// TwinCAT 3 PLC project tc_project_app
// ProgramVersion: 3.1.4023.0
// libraries:
//   Tc2_EtherCAT, * (Beckhoff Automation GmbH)
//   Tc2_MC2, * (Beckhoff Automation GmbH)
//   Tc2_MC2_Drive, * (Beckhoff Automation GmbH)
//   Tc2_Standard, * (Beckhoff Automation GmbH)
//   Tc2_SUPS, * (Beckhoff Automation GmbH)
//   Tc2_System, * (Beckhoff Automation GmbH)
//   Tc2_Utilities, * (Beckhoff Automation GmbH)
//   Tc3_MC2_AdvancedHoming, * (Beckhoff Automation GmbH)
//   Tc3_Module, * (Beckhoff Automation GmbH)
//   VisuDialogs, * (System)
// project tree:
//   DUTs/ E_RotationBrakeCheckerState.TcDUT, ST_AxisSpg.TcDUT, ST_DefaultVals.TcDUT
//   / GlobalTextList.TcGTLO (not stored), PlcTask.TcTTO, Visualization Manager.TcVMO (not stored)
//   GVLs/ GVL_APP.TcGVL, GVL_INTER.TcGVL, GVL_Safety.TcGVL
//   POUs/Application_Specific/Applications/ Application_Template.TcPOU (not stored), eState_INTER.TcDUT, eState_Vertical.TcDUT, Inclinometer.TcPOU, INTER_LOGIC.TcPOU, PLC_SAFETY_LOGIC.TcPOU, SBT_CODE_notused.TcPOU, Slit_3.TcPOU, VirtualSpeedOverrides.TcPOU
//   POUs/Application_Specific/Axes/ AXIS_NAMES.TcGVL, Axis_Template.TcPOU (not stored), Slit_West.TcPOU, Slit_North.TcPOU, Combined_Vertical.TcPOU, Horizontal_Translation.TcPOU, Slit_South.TcPOU, Slit_East.TcPOU, Vertical_Translation_Y2.TcPOU, Vertical_Translation_Y1.TcPOU, Rotation.TcPOU, Pneumatics_Template.TcPOU (not stored)
//   POUs/Application_Specific/Axes/Real axis follows/ Combined_Vertical_Virtual.TcPOU, Horizontal_Virtual.TcPOU, Rotation_Virtual.TcPOU
//   POUs/Application_Specific/Axes/Sample and Calibration/ Measurement_Angle_Offset.TcPOU, Rotation_Calibration.TcPOU, Horizontal_Calibration.TcPOU, Combined_Vertical_Calibration.TcPOU, Rotation_Sample.TcPOU, Horizontal_Sample.TcPOU, Combined_Vertical_Sample.TcPOU
//   POUs/Application_Specific/Axes/Virtuals/ Delta.TcPOU, Doff_Angled.TcPOU, Doff_Parallel.TcPOU, Drad.TcPOU, Drad_External.TcPOU, Drad_Internal.TcPOU, Dtank_Internal_Offset_Angle.TcPOU, Dtank_Length.TcPOU, Dtank_Pivot_To_Window.TcPOU, Measurement_Angle.TcPOU, Tau.TcPOU
//   POUs/ MAIN.TcPOU
//   tc_mca_std_lib/DUTs/Axis_Structures/ ST_AxisConfig.TcDUT (not stored), ST_AxisControl.TcDUT (not stored), ST_AxisDescription.TcDUT, ST_AxisError.TcDUT (not stored), ST_AxisInputs.TcDUT (not stored), ST_AxisPersistent.TcDUT (not stored), ST_AxisSafety.TcDUT (not stored), ST_AxisStatus.TcDUT, ST_AxisStruct.TcDUT, ST_GearAxis.TcDUT (not stored)
//   tc_mca_std_lib/DUTs/ E_AxisParameters.TcTLEO (not stored), E_HomingRoutines.TcTLEO, E_AxisParameters.TcTLEO (not stored), E_MonitoringLedFunction.TcDUT (not stored), E_MotorTypeClass.TcDUT, E_EncoderTypeClass.TcDUT, E_HomeSwitchTypeClass.TcDUT, E_RestorePosition.TcDUT (not stored), I_Axis.TcIO (not stored), E_SlitPairStatesV2.TcDUT (not stored), E_SlitPairStates.TcDUT (not stored), ST_MonitoringAlarm.TcDUT (not stored), E_MotionFunctions.TcDUT (not stored), ST_McStatus.TcDUT (not stored)
//   tc_mca_std_lib/DUTs/Pneumatics/ E_PneumaticAxisErrors.TcDUT (not stored), E_PneumaticMode.TcDUT (not stored), ST_PneumaticAxisControl.TcDUT (not stored), ST_PneumaticAxisConfig.TcDUT (not stored), ST_PneumaticAxisInputs.TcDUT (not stored), ST_PneumaticAxisOutputs.TcDUT (not stored), ST_PneumaticAxisStatus.TcDUT (not stored), ST_PneumaticAxisStruct.TcDUT (not stored)
//   tc_mca_std_lib/DUTs/Safety Status/ E_SafetyFbState.TcDUT, E_SafetyFbType.TcDUT, E_SafetyGroupState.TcDUT, E_SafetyDevices.TcDUT (not stored), FB_SafeFBDiag.TcPOU, ST_SafetyAliasInput.TcDUT, ST_SafetyData.TcDUT, ST_SafetyDevice.TcDUT (not stored), ST_SafetyFB.TcDUT, ST_SafetyGroup.TcDUT, ST_SafetyAliasOutput.TcDUT, ST_SafetyProject.TcDUT
//   tc_mca_std_lib/GVLs/ GVL.TcGVL
//   tc_mca_std_lib/POUs/ FB_ESSMonitoring.TcPOU
//   tc_mca_std_lib/POUs/Motion/ FB_Axis.TcPOU, FB_SlitPair.TcPOU (not stored), FB_SlitPairV2.TcPOU (not stored)
//   tc_mca_std_lib/POUs/Motion/Homing/ FB_Homing.TcPOU (not stored)
//   tc_mca_std_lib/POUs/Pneumatics/ FB_PneumaticAxis.TcPOU (not stored)
//   tc_mca_std_lib/VISUs/ languageSupport.TcTLO (not stored), MainVisu.TcVIS, ParameterTextList.TcTLO (not stored), PneumaticsVisu.TcVIS (not stored)
// real-time tasks:
//   TASK PlcTask: cycle T#2ms, priority 10, ADS port 351
// motion (NC):
//   TASK NC-Task 1 SAF: cycle T#2ms, priority 4, ADS port 501
//   TASK NC-Task 1 SVB: cycle T#10ms, priority 8, ADS port 511
//   AXIS M1 - South (id 1)
//     Dynamic: AccelerationMaximum=50, DecelerationMaximum=50, Acceleration=25, Deceleration=25, Jerk=60
//     Velo: RefSearch=0.5, RefSync=0.5, SlowManual=0.5, FastManual=1, Maximum=1.2
//     OtherSettings: AllowMotionCmdToSlave=true, DataPersistence=true
//     encoder EncType=4
//       EncPara: ScaleFactorNumerator=0.001, MaxCount=#x0000ffff
//         Inc: RefMode=2, RefSoftSyncMask=#x0000ffff
//     drive DrvType=24
//       DrvPara: Inverse=true
//         Analog: VeloReferenz=2, TorqueSetpointScale=10, ScaleFactorActTorque=0.1
//         TimeComp: TaskDelayCycles=1
//     controller CtrType=1
//       CtrPara: PriorControlFactor=1
//         Observer: BandWidth=20
//   AXIS M2 - North (id 2)
//     Dynamic: AccelerationMaximum=50, DecelerationMaximum=50, Acceleration=25, Deceleration=25, Jerk=60
//     Velo: RefSearch=0.5, RefSync=0.5, SlowManual=0.5, FastManual=1, Maximum=1.2
//     OtherSettings: AllowMotionCmdToSlave=true, DataPersistence=true
//     encoder EncType=4
//       EncPara: ScaleFactorNumerator=0.001, MaxCount=#x0000ffff
//         Inc: RefMode=2, RefSoftSyncMask=#x0000ffff
//     drive DrvType=24
//       Analog: VeloReferenz=2, TorqueSetpointScale=10, ScaleFactorActTorque=0.1
//       TimeComp: TaskDelayCycles=1
//     controller CtrType=1
//       CtrPara: PriorControlFactor=1
//         Observer: BandWidth=20
//   AXIS M3 - West (id 3)
//     Dynamic: AccelerationMaximum=50, DecelerationMaximum=50, Acceleration=25, Deceleration=25, Jerk=60
//     Velo: RefSearch=0.5, RefSync=0.5, SlowManual=0.5, FastManual=1, Maximum=1.2
//     OtherSettings: AllowMotionCmdToSlave=true, DataPersistence=true
//     encoder EncType=4
//       EncPara: ScaleFactorNumerator=0.001, MaxCount=#x0000ffff
//         Inc: RefMode=2, RefSoftSyncMask=#x0000ffff
//     drive DrvType=24
//       DrvPara: Inverse=true
//         Analog: VeloReferenz=2, TorqueSetpointScale=10, ScaleFactorActTorque=0.1
//         TimeComp: TaskDelayCycles=1
//     controller CtrType=1
//       CtrPara: PriorControlFactor=1
//         Observer: BandWidth=20
//   AXIS M4 - East (id 4)
//     Dynamic: AccelerationMaximum=50, DecelerationMaximum=50, Acceleration=25, Deceleration=25, Jerk=60
//     Velo: RefSearch=0.5, RefSync=0.5, SlowManual=0.5, FastManual=1, Maximum=1.2
//     OtherSettings: AllowMotionCmdToSlave=true, DataPersistence=true
//     encoder EncType=4
//       EncPara: ScaleFactorNumerator=0.001, MaxCount=#x0000ffff
//         Inc: RefMode=2, RefSoftSyncMask=#x0000ffff
//     drive DrvType=24
//       Analog: VeloReferenz=2, TorqueSetpointScale=10, ScaleFactorActTorque=0.1
//       TimeComp: TaskDelayCycles=1
//     controller CtrType=1
//       CtrPara: PriorControlFactor=1
//         Observer: BandWidth=20
//   AXIS Rotation (id 5)
//     General: UnitName=°
//     Dynamic: AccelerationMaximum=19997.325, DecelerationMaximum=19997.325, Acceleration=30, Deceleration=30, Jerk=35.7075
//     Velo: RefSearch=0.07935, RefSync=0.07935, SlowManual=0.05, FastManual=0.6, Fast=7.935, Maximum=8
//     OtherSettings: AllowMotionCmdToSlave=true, DataPersistence=true
//     encoder EncType=19
//       EncPara: ScaleFactorNumerator=360, ScaleFactorDenominator=1761607680, Offset=-201.549349812099, MaxCount=#xffffffff, ReferenceSystem=1
//     drive DrvType=16
//       DrvPara: MaxCount=#xffffffff, DriveControlDWord=#x00020100
//         Analog: VeloReferenz=8.7285, VeloScale=71.5255737304688, TorqueSetpointScale=10, ScaleFactorActTorque=0.1
//         TimeComp: TaskDelayCycles=1
//     controller CtrType=1
//       CtrPara: PriorControlFactor=1
//         PosDiffControl: Range=4
//         Observer: BandWidth=20
//   AXIS Horizontal Z Translation (id 6)
//     Dynamic: Acceleration=34.773, Deceleration=34.773, Jerk=104.319
//     Velo: RefSearch=0.23182, RefSync=0.23182, SlowManual=2, FastManual=4, Fast=23.182, Maximum=20
//     PositionAreaControl: Enable=false
//     TargetPosControl: Range=0.005, Time=0.04
//     OtherSettings: AllowMotionCmdToSlave=true
//     encoder EncType=19
//       EncPara: ScaleFactorNumerator=0.001, ScaleFactorDenominator=1000, Offset=2359.51, Inverse=true, MaxCount=#xffffffff, ReferenceSystem=1
//         Inc: RefSoftSyncMask=#x0007a11f
//     drive DrvType=16
//       DrvPara: Inverse=true, MaxCount=#xffffffff, DriveControlDWord=#x00020000
//         Analog: VeloReferenz=25.5002, VeloScale=71.5255737304688, TorqueSetpointScale=10, ScaleFactorActTorque=0.1
//         TimeComp: TaskDelayCycles=1
//     controller CtrType=1
//       CtrPara: PriorControlFactor=1
//         PosDiffControl: Enable=false
//         Observer: BandWidth=20
//   AXIS Vertical Y1 (id 7) // ACTUALLY Y?
//     Dynamic: Acceleration=10, Deceleration=10, Jerk=40
//     Velo: RefSearch=0.37029, RefSync=0.37029, SlowManual=5, FastManual=30, Fast=37.029, Maximum=32
//     PositionAreaControl: Enable=false
//     TargetPosControl: Range=0.01
//     OtherSettings: AllowMotionCmdToSlave=true
//     encoder EncType=19
//       EncPara: ScaleFactorNumerator=0.001, ScaleFactorDenominator=1000, Offset=91.510823, Inverse=true, MaxCount=#xffffffff, ReferenceSystem=1, EncPositionSource=1
//         Inc: RefSoftSyncMask=#x000f423f
//     drive DrvType=16
//       DrvPara: Inverse=true, MaxCount=#xffffffff, DriveControlDWord=#x00020000
//         Analog: VeloReferenz=40.7319, VeloScale=71.5255737304688, TorqueSetpointScale=10, ScaleFactorActTorque=0.1
//         TimeComp: TaskDelayCycles=1
//     controller CtrType=1
//       CtrPara: PriorControlFactor=1
//         PID: PosKp=2
//         Observer: BandWidth=20
//   AXIS Vertical Y2 (id 8)
//     Dynamic: Acceleration=10, Deceleration=10, Jerk=40
//     Velo: RefSearch=0.37029, RefSync=0.37029, SlowManual=5, FastManual=30, Fast=37.029, Maximum=32
//     PositionAreaControl: Enable=false
//     TargetPosControl: Range=0.01
//     OtherSettings: AllowMotionCmdToSlave=true
//     encoder EncType=19
//       EncPara: ScaleFactorNumerator=0.001, ScaleFactorDenominator=1000, Offset=93.490647, MaxCount=#xffffffff, ReferenceSystem=1
//         Inc: RefSoftSyncMask=#x000f423f
//     drive DrvType=16
//       DrvPara: MaxCount=#xffffffff, DriveControlDWord=#x00020000
//         Analog: VeloReferenz=40.7319, VeloScale=71.5255737304688, TorqueSetpointScale=10, ScaleFactorActTorque=0.1
//         TimeComp: TaskDelayCycles=1
//     controller CtrType=1
//       CtrPara: PriorControlFactor=1
//         PID: PosKp=2
//         Observer: BandWidth=20
//   AXIS RotExtra (id 31)
//     OtherSettings: AllowMotionCmdToSlave=true
//     encoder EncType=16
//       EncPara: ScaleFactorNumerator=360, ScaleFactorDenominator=1761607680, MaxCount=#xffffffff
//     drive DrvType=5
//       Analog: TorqueSetpointScale=10, ScaleFactorActTorque=0.1
//       TimeComp: TaskDelayCycles=1
//     controller CtrType=1
//       CtrPara: PriorControlFactor=1
//         Observer: BandWidth=20
//   AXIS Detector Tank Internal Offset Angle (id 14)
//     OtherSettings: AllowMotionCmdToSlave=true
//     encoder EncType=16
//       EncPara: ScaleFactorNumerator=1e-05, MaxCount=#xffffffff, ReferenceSystem=1
//     drive DrvType=5
//       Analog: TorqueSetpointScale=10, ScaleFactorActTorque=0.1
//       TimeComp: TaskDelayCycles=1
//     controller CtrType=1
//       CtrPara: PriorControlFactor=1
//         Observer: BandWidth=20
//   AXIS Delta (id 17)
//     OtherSettings: AllowMotionCmdToSlave=true
//     encoder EncType=16
//       EncPara: ScaleFactorNumerator=1e-05, MaxCount=#xffffffff, ReferenceSystem=1
//     drive DrvType=5
//       Analog: TorqueSetpointScale=10, ScaleFactorActTorque=0.1
//       TimeComp: TaskDelayCycles=1
//     controller CtrType=1
//       CtrPara: PriorControlFactor=1
//         Observer: BandWidth=20
//   AXIS Tau (id 18)
//     OtherSettings: AllowMotionCmdToSlave=true
//     encoder EncType=16
//       EncPara: ScaleFactorNumerator=1e-05, MaxCount=#xffffffff, ReferenceSystem=1
//     drive DrvType=5
//       Analog: TorqueSetpointScale=10, ScaleFactorActTorque=0.1
//       TimeComp: TaskDelayCycles=1
//     controller CtrType=1
//       CtrPara: PriorControlFactor=1
//         Observer: BandWidth=20
//   AXIS Detector Radius External (id 10)
//     OtherSettings: AllowMotionCmdToSlave=true
//     encoder EncType=16
//       EncPara: ScaleFactorNumerator=1e-05, MaxCount=#xffffffff, ReferenceSystem=1
//     drive DrvType=5
//       Analog: TorqueSetpointScale=10, ScaleFactorActTorque=0.1
//     controller CtrType=1
//       CtrPara: PriorControlFactor=1
//         Observer: BandWidth=20
//   AXIS Detector Radius Internal (id 11)
//     OtherSettings: AllowMotionCmdToSlave=true
//     encoder EncType=16
//       EncPara: ScaleFactorNumerator=1e-05, MaxCount=#xffffffff, ReferenceSystem=1
//     drive DrvType=5
//       Analog: TorqueSetpointScale=10, ScaleFactorActTorque=0.1
//     controller CtrType=1
//       CtrPara: PriorControlFactor=1
//         Observer: BandWidth=20
//   AXIS Combined Vertical (id 9)
//     Dynamic: Acceleration=60, Deceleration=60, Jerk=40
//     Velo: RefSearch=0.37029, RefSync=0.37029, SlowManual=10, FastManual=15, Fast=37.029, Maximum=30
//     PositionAreaControl: Enable=false
//     TargetPosControl: Range=0.005, Time=0.2
//     OtherSettings: AllowMotionCmdToSlave=true
//     encoder EncType=1
//       EncPara: ScaleFactorNumerator=0.001, ScaleFactorDenominator=1000, Offset=67.6442, Inverse=true, ReferenceSystem=1
//     drive DrvType=5
//       DrvPara: Inverse=true
//         Analog: VeloReferenz=40.7319, TorqueSetpointScale=10, ScaleFactorActTorque=0.1
//         TimeComp: TaskDelayCycles=1
//     controller CtrType=1
//       CtrPara: PriorControlFactor=0.8
//         Observer: BandWidth=20
//   AXIS Horizontal Virtual (id 30)
//     OtherSettings: AllowMotionCmdToSlave=true
//     encoder EncType=16
//       EncPara: ScaleFactorNumerator=1e-05, MaxCount=#xffffffff, ReferenceSystem=1
//     drive DrvType=5
//       Analog: TorqueSetpointScale=10, ScaleFactorActTorque=0.1
//       TimeComp: TaskDelayCycles=1
//     controller CtrType=1
//       CtrPara: PriorControlFactor=1
//         Observer: BandWidth=20
//   AXIS Rotation Virtual (id 23)
//     OtherSettings: AllowMotionCmdToSlave=true
//     encoder EncType=16
//       EncPara: ScaleFactorNumerator=1e-05, MaxCount=#xffffffff, ReferenceSystem=1
//     drive DrvType=5
//       Analog: TorqueSetpointScale=10, ScaleFactorActTorque=0.1
//       TimeComp: TaskDelayCycles=1
//     controller CtrType=1
//       CtrPara: PriorControlFactor=1
//         Observer: BandWidth=20
//   AXIS Combined Vertical Virtual (id 27)
//     OtherSettings: AllowMotionCmdToSlave=true
//     encoder EncType=16
//       EncPara: ScaleFactorNumerator=1e-05, MaxCount=#xffffffff, ReferenceSystem=1
//     drive DrvType=5
//       Analog: TorqueSetpointScale=10, ScaleFactorActTorque=0.1
//       TimeComp: TaskDelayCycles=1
//     controller CtrType=1
//       CtrPara: PriorControlFactor=1
//         Observer: BandWidth=20
//   AXIS Detector Tank Length (id 15)
//     Dynamic: Acceleration=20, Deceleration=20, Jerk=50
//     Velo: SlowManual=5, FastManual=10
//     OtherSettings: AllowMotionCmdToSlave=true
//     encoder EncType=1
//     drive DrvType=5
//       Analog: TorqueSetpointScale=10, ScaleFactorActTorque=0.1
//       TimeComp: TaskDelayCycles=1
//     controller CtrType=1
//       CtrPara: PriorControlFactor=1
//         Observer: BandWidth=20
//   AXIS Detector Tank Pivot To Window (id 16)
//     Dynamic: Acceleration=20, Deceleration=20, Jerk=50
//     Velo: SlowManual=5, FastManual=10
//     OtherSettings: AllowMotionCmdToSlave=true
//     encoder EncType=1
//     drive DrvType=5
//       Analog: TorqueSetpointScale=10, ScaleFactorActTorque=0.1
//       TimeComp: TaskDelayCycles=1
//     controller CtrType=1
//       CtrPara: PriorControlFactor=1
//         Observer: BandWidth=20
//   AXIS Rotation Calibration (id 22)
//     General: UnitName=°
//     Dynamic: Acceleration=0.5, Deceleration=0.5, Jerk=30
//     Velo: RefSearch=0.55548, RefSync=0.55548, SlowManual=0.25, FastManual=0.375, Fast=55.543, Maximum=55.543
//     TargetPosControl: Range=0.005
//     OtherSettings: AllowMotionCmdToSlave=true, DataPersistence=true
//     encoder EncType=1
//       EncPara: ScaleFactorNumerator=360, ScaleFactorDenominator=251658240, Offset=10.2575826644897, ToleranceWndModuloStart=10
//     drive DrvType=5
//       Analog: VeloReferenz=61.0973, TorqueSetpointScale=10, ScaleFactorActTorque=0.1
//       TimeComp: TaskDelayCycles=1
//     controller CtrType=1
//       CtrPara: PriorControlFactor=1
//         PID: PosKp=2
//         Observer: BandWidth=20
//   AXIS Combined Vertical Calibration (id 25)
//     Dynamic: Acceleration=20, Deceleration=20, Jerk=50
//     Velo: SlowManual=5, FastManual=10, Fast=37.029, Maximum=37.029
//     PositionAreaControl: Enable=false
//     TargetPosControl: Range=0.005, Time=0.2
//     OtherSettings: AllowMotionCmdToSlave=true
//     encoder EncType=1
//       EncPara: ScaleFactorNumerator=0.001, ScaleFactorDenominator=1000, Offset=182.9435, Inverse=true, ReferenceSystem=1
//     drive DrvType=5
//       DrvPara: Inverse=true
//         Analog: VeloReferenz=40.7319, TorqueSetpointScale=10, ScaleFactorActTorque=0.1
//         TimeComp: TaskDelayCycles=1
//     controller CtrType=1
//       CtrPara: PriorControlFactor=0.8
//         Observer: BandWidth=20
//   AXIS Horizontal Calibration (id 28)
//     Dynamic: Acceleration=20, Deceleration=20, Jerk=50
//     Velo: SlowManual=5, FastManual=10, Fast=23.182, Maximum=23.182
//     PositionAreaControl: Enable=false
//     TargetPosControl: Range=0.005, Time=0.04
//     OtherSettings: AllowMotionCmdToSlave=true
//     encoder EncType=1
//       EncPara: ScaleFactorNumerator=5, ScaleFactorDenominator=10485760, Offset=2359.51, ModuloFactor=100000000, Inverse=true, EncPositionSource=1
//     drive DrvType=5
//       DrvPara: Inverse=true
//         Analog: VeloReferenz=25.5002, TorqueSetpointScale=10, ScaleFactorActTorque=0.1
//         TimeComp: TaskDelayCycles=1
//     controller CtrType=1
//       CtrPara: PriorControlFactor=1
//         PID: PosKp=2
//         Observer: BandWidth=20
//   AXIS Detector Offset Angled (id 12)
//     Dynamic: Acceleration=0.5, Deceleration=0.5, Jerk=30
//     Velo: RefSearch=0.55548, RefSync=0.55548, SlowManual=0.25, FastManual=0.375
//     OtherSettings: AllowMotionCmdToSlave=true
//     encoder EncType=1
//     drive DrvType=5
//       Analog: TorqueSetpointScale=10, ScaleFactorActTorque=0.1
//       TimeComp: TaskDelayCycles=1
//     controller CtrType=1
//       CtrPara: PriorControlFactor=1
//         Observer: BandWidth=20
//   AXIS Detector Offset Parallel (id 13)
//     Dynamic: Acceleration=0.5, Deceleration=0.5, Jerk=30
//     Velo: RefSearch=0.55548, RefSync=0.55548, SlowManual=5, FastManual=10
//     OtherSettings: AllowMotionCmdToSlave=true
//     encoder EncType=1
//     drive DrvType=5
//       Analog: TorqueSetpointScale=10, ScaleFactorActTorque=0.1
//       TimeComp: TaskDelayCycles=1
//     controller CtrType=1
//       CtrPara: PriorControlFactor=1
//         Observer: BandWidth=20
//   AXIS Detector Radius (id 19)
//     Dynamic: Acceleration=20, Deceleration=20, Jerk=50
//     Velo: SlowManual=5, FastManual=10
//     OtherSettings: AllowMotionCmdToSlave=true
//     encoder EncType=1
//       EncPara: ScaleFactorNumerator=1e-06
//     drive DrvType=5
//       Analog: TorqueSetpointScale=10, ScaleFactorActTorque=0.1
//       TimeComp: TaskDelayCycles=1
//     controller CtrType=1
//       CtrPara: PriorControlFactor=1
//         Observer: BandWidth=20
//   AXIS Measurement Angle (id 20)
//     Dynamic: AccelerationMaximum=600, DecelerationMaximum=600, Acceleration=0.3, Deceleration=0.3, Jerk=10
//     Velo: RefSearch=0.55548, RefSync=0.55548, SlowManual=0.25, FastManual=0.375, Maximum=2
//     OtherSettings: AllowMotionCmdToSlave=true
//     encoder EncType=1
//       EncPara: ScaleFactorNumerator=1e-06
//     drive DrvType=5
//       Analog: TorqueSetpointScale=10, ScaleFactorActTorque=0.1
//       TimeComp: TaskDelayCycles=1
//     controller CtrType=1
//       CtrPara: PriorControlFactor=1
//         Observer: BandWidth=20
//   AXIS Measurement Angle Offset (id 21)
//     Dynamic: AccelerationMaximum=600, DecelerationMaximum=600, Acceleration=0.5, Deceleration=0.5, Jerk=30
//     Velo: RefSearch=0.55548, RefSync=0.55548, SlowManual=0.25, FastManual=0.375, Maximum=0.6
//     OtherSettings: AllowMotionCmdToSlave=true
//     encoder EncType=1
//       EncPara: ScaleFactorNumerator=1e-06
//     drive DrvType=5
//       Analog: TorqueSetpointScale=10, ScaleFactorActTorque=0.1
//       TimeComp: TaskDelayCycles=1
//     controller CtrType=1
//       CtrPara: PriorControlFactor=1
//         Observer: BandWidth=20
//   AXIS Rotation Sample (id 24)
//     General: UnitName=°
//     Dynamic: Acceleration=0.5, Deceleration=0.5, Jerk=30
//     Velo: RefSearch=0.55548, RefSync=0.55548, SlowManual=0.25, FastManual=0.375, Fast=55.543, Maximum=55.543
//     OtherSettings: AllowMotionCmdToSlave=true, DataPersistence=true
//     encoder EncType=1
//       EncPara: ScaleFactorNumerator=360, ScaleFactorDenominator=251658240, Offset=10.2575826644897, ToleranceWndModuloStart=10
//     drive DrvType=5
//       Analog: VeloReferenz=61.0973, TorqueSetpointScale=10, ScaleFactorActTorque=0.1
//       TimeComp: TaskDelayCycles=1
//     controller CtrType=1
//       CtrPara: PriorControlFactor=1
//         PID: PosKp=2
//         Observer: BandWidth=20
//   AXIS Combined Vertical Sample (id 26)
//     Dynamic: Acceleration=20, Deceleration=20, Jerk=50
//     Velo: SlowManual=5, FastManual=10, Fast=37.029, Maximum=37.029
//     PositionAreaControl: Enable=false
//     TargetPosControl: Range=0.005, Time=0.2
//     OtherSettings: AllowMotionCmdToSlave=true
//     encoder EncType=1
//       EncPara: ScaleFactorNumerator=0.001, ScaleFactorDenominator=1000, Inverse=true, ReferenceSystem=1
//     drive DrvType=5
//       DrvPara: Inverse=true
//         Analog: VeloReferenz=40.7319, TorqueSetpointScale=10, ScaleFactorActTorque=0.1
//         TimeComp: TaskDelayCycles=1
//     controller CtrType=1
//       CtrPara: PriorControlFactor=0.8
//         Observer: BandWidth=20
//   AXIS Horizontal Sample (id 29)
//     Dynamic: Acceleration=34.773, Deceleration=34.773, Jerk=104.319
//     Velo: RefSearch=0.23182, RefSync=0.23182, SlowManual=5, FastManual=10, Fast=23.182, Maximum=23.182
//     PositionAreaControl: Enable=false
//     TargetPosControl: Range=0.005, Time=0.04
//     OtherSettings: AllowMotionCmdToSlave=true
//     encoder EncType=1
//       EncPara: ScaleFactorNumerator=5, ScaleFactorDenominator=10485760, Offset=2359.51, ModuloFactor=100000000, Inverse=true, EncPositionSource=1
//     drive DrvType=5
//       DrvPara: Inverse=true
//         Analog: VeloReferenz=25.5002, TorqueSetpointScale=10, ScaleFactorActTorque=0.1
//         TimeComp: TaskDelayCycles=1
//     controller CtrType=1
//       CtrPara: PriorControlFactor=1
//         PID: PosKp=2
//         Observer: BandWidth=20
// I/O:
//   DEVICE Device 1 (EtherCAT), AmsNetId 5.119.206.217.2.1
//     Term 1 (EK1200) [EK1200-5000 EtherCAT Power supply (2A E-Bus)]
//       Term 2 (EL6070-0033) [EL6070-0033 1Ch. Licence key terminal, individual licences]
//       Term 3 (EL3004) [EL3004 4Ch. Ana. Input +/-10V]
//       Term 39 (EL3621-0020) [EL3621-0020 1Ch. Ana. Input 4-20 mA, Diff. 24bit, High Precision, calibrated]
//       Term 5 (EL4004) [EL4004 4Ch. Ana. Output 0-10V, 12bit]
//       Term 6 (EL4024) [EL4024 4Ch. Ana. Output 4-20mA, 12bit]
//       Term 7 (EL1008) [EL1008 8Ch. Dig. Input 24V, 3ms]
//       Term 8 (EL2008) [EL2008 8Ch. Dig. Output 24V, 0.5A]
//       Term 9 (EL1008) [EL1008 8Ch. Dig. Input 24V, 3ms]
//       EL10088-(03) [EL1008 8Ch. Dig. Input 24V, 3ms]
//       Term 11 (EL6688) [EL6688 - External Synchronisation Interface (IEEE1588)]
//       Term 12 (EL9410) [EL9410 E-Bus Power Supplier  (Diagnostics)]
//       EL2008-(02) [EL2008 8Ch. Dig. Output 24V, 0.5A]
//       EL2008-(03) [EL2008 8Ch. Dig. Output 24V, 0.5A]
//       Term 50 (EL3152) [EL3152 2Ch. Ana Input 4-20mA]
//       Term 16 (EK1110) [EK1110 EtherCAT extension]
//     Term 17 (EK1100) [EK1100 EtherCAT Coupler (2A E-Bus)]
//       Term 18 (EL5101) [EL5101 1Ch. Inc. Encoder 5V]
//       Term 19 (EL5101) [EL5101 1Ch. Inc. Encoder 5V]
//       Term 20 (EL5101) [EL5101 1Ch. Inc. Encoder 5V]
//       Term 21 (EL5101) [EL5101 1Ch. Inc. Encoder 5V]
//       Term 36 (EL9011) [EL9011 End Terminal]
//     Term 22 (EK1100) [EK1100 EtherCAT Coupler (2A E-Bus)]
//       Term 23 (EL7047) [EL7047 1Ch. Stepper motor output stage (50V, 5A)]
//       Term 24 (EL7047) [EL7047 1Ch. Stepper motor output stage (50V, 5A)]
//       Term 25 (EL7047) [EL7047 1Ch. Stepper motor output stage (50V, 5A)]
//       Term 26 (EL7047) [EL7047 1Ch. Stepper motor output stage (50V, 5A)]
//       Term 37 (EL9011) [EL9011 End Terminal]
//     Term 27 (EK1100) [EK1100 EtherCAT Coupler (2A E-Bus)]
//       EL6910-(04) [EL6910, TwinSAFE PLC]
//       EL2904-(06) [EL2904, 4 Ch. Safety Output 24V, 0.5A, TwinSAFE]
//         modules: Module 1 (FSOES), Module 2 (DO)
//       EL1904-(06) [EL1904, 4 Ch. Safety Input 24V, TwinSAFE]
//         modules: Module 1 (FSOES)
//       EL1904-(07) [EL1904, 4 Ch. Safety Input 24V, TwinSAFE]
//         modules: Module 1 (FSOES)
//       EL1904-(08) [EL1904, 4 Ch. Safety Input 24V, TwinSAFE]
//         modules: Module 1 (FSOES)
//       EL1904-(09) [EL1904, 4 Ch. Safety Input 24V, TwinSAFE]
//         modules: Module 1 (FSOES)
//       EL1904-(10) [EL1904, 4 Ch. Safety Input 24V, TwinSAFE]
//         modules: Module 1 (FSOES)
//       EL1904-(11) [EL1904, 4 Ch. Safety Input 24V, TwinSAFE]
//         modules: Module 1 (FSOES)
//       EL2912-(07) [EL2912, 2Ch. Safety Output 24V, 2A, TwinSAFE]
//         modules: Module 1 (FSOE), Module 2 (FSOUT), Module 3 (DEVICEIO), Module 4 (FSLOGIC)
//       Term 80 (EL9410) [EL9410 E-Bus Power Supplier  (Diagnostics)]
//       EL1904-(12) [EL1904, 4 Ch. Safety Input 24V, TwinSAFE]
//         modules: Module 1 (FSOES)
//       EL1904-(13) [EL1904, 4 Ch. Safety Input 24V, TwinSAFE]
//         modules: Module 1 (FSOES)
//       EL2904-(08) [EL2904, 4 Ch. Safety Output 24V, 0.5A, TwinSAFE]
//         modules: Module 1 (FSOES), Module 2 (DO)
//       EL2904-(09) [EL2904, 4 Ch. Safety Output 24V, 0.5A, TwinSAFE]
//         modules: Module 1 (FSOES), Module 2 (DO)
//       Term 38 (EL9011) [EL9011 End Terminal]
//     Term 70 (AX8640-0000-0103) [AX8640-0000-0103]
//       Drive 71 (AX8206-0210-0104) [AX8206-0210-0104 (2Ch. 6A servo axis, safe-motion, multi-FB)]
//         modules: Device, Device, Device, Device, Device, Device, Device, Device, Device, Device, Device (Safety), Device, Device, Device, Device, Device, Device, Device, Device, Device, Device, Device, Device, Device, Device, Device, Device, Device, Device, Device, Device, Ch A, Ch A, Ch A, Ch A, Ch A, Ch A, Ch A, Ch A, Ch A, Ch A, Ch A, Ch A, Ch A, Ch A, Ch A, Ch A, Ch A, Ch A, Ch A, Ch A, Ch A, Ch A, Ch A, Ch A, Ch A, Ch A, Ch A, Ch B, Ch B, Ch B, Ch B, Ch B, Ch B, Ch B, Ch B, Ch B, Ch B, Ch B, Ch B, Ch B, Ch B, Ch B, Ch B, Ch B, Ch B, Ch B, Ch B, Ch B, Ch B, Ch B, Ch B, Ch B, Ch B, Ch B
//         startup 12992:1 := 414D383035332D78477831 // Ch A Motor parameters / Configured motor type
//         startup 24768:0 := FEFF // Ch A Interpolation sub mode select
//         startup 13000:5 := 0200 // Ch A Motor thermal model / Reaction
//         startup 13000:6 := 0000C841 // Ch A Motor thermal model / Partial fraction factor
//         startup 12992:12 := 0000FA44 // Ch A Motor parameters / Motor rated speed
//         startup 12992:13 := 73681F41 // Ch A Motor parameters / Motor rated torque
//         startup 24694:0 := 9D2C0000 // Ch A Motor standstill torque
//         startup 24800:0 := D007 // Ch A Positive torque/force limit value
//         startup 24801:0 := D007 // Ch A Negative torque/force limit value
//         startup 12288:6 := 4158383230362D303231302D30303030 // Ch A AxisMain parameters / Configured drive type
//         startup 12867:1 := 66669640 // Ch A TorqueCtrl parameters / Configured channel rated current
//         startup 12867:2 := 9A996141 // Ch A TorqueCtrl parameters / Configured channel peak current
//         startup 24672:0 := 08 // Ch A Modes of operation
//         startup 12864:1 := 0501AA42 // Ch A TorqueCtrl parameters mappable / Torque control proportional gain q
//         startup 12864:2 := 8A0E7C39 // Ch A TorqueCtrl parameters mappable / Torque control integral action time q
//         startup 12608:1 := F6F4A83E // Ch A VeloCtrl parameters mappable / Velocity control proportional gain
//         startup 12608:2 := 6F12033C // Ch A VeloCtrl parameters mappable / Velocity control integral action time
//         startup 12608:3 := 00980546 // Ch A VeloCtrl parameters mappable / Bipolar velocity limit value
//         startup 12992:15 := 0100 // Ch A Motor parameters / Motor temperature sensor connection
//         startup 12611:4 := 0400 // Ch A VeloCtrl observer / Observer type
//         startup 24672:0 := 08 // Ch A Modes of operation
//         startup 12296:2 := 00 // Ch A AxisMain parameters encoder polarity / Primary encoder actual values
//         startup 12611:4 := 0400 // Ch A VeloCtrl observer / Observer type
//         startup 13071:2 := 00000000 // Ch A Secondary Feedback BiSS-C: Encoder parameter (rotary) / Power supply
//         startup 13071:5 := 00 // Ch A Secondary Feedback BiSS-C: Encoder parameter (rotary) / Data layout
//         startup 13071:6 := 00 // Ch A Secondary Feedback BiSS-C: Encoder parameter (rotary) / Fill bit count left
//         startup 13071:7 := 00 // Ch A Secondary Feedback BiSS-C: Encoder parameter (rotary) / Fill bit count right
//         startup 12296:1 := 00 // Ch A AxisMain parameters encoder polarity / Secondary encoder actual values
//         startup 14016:1 := 414D383034332D78457831 // Ch B Motor parameters / Configured motor type
//         startup 26816:0 := FEFF // Ch B Interpolation sub mode select
//         startup 14024:5 := 0200 // Ch B Motor thermal model / Reaction
//         startup 14016:12 := 00401C45 // Ch B Motor parameters / Motor rated speed
//         startup 14016:13 := E17AA840 // Ch B Motor parameters / Motor rated torque
//         startup 26742:0 := 17160000 // Ch B Motor standstill torque
//         startup 26848:0 := D007 // Ch B Positive torque/force limit value
//         startup 26849:0 := D007 // Ch B Negative torque/force limit value
//         startup 13312:6 := 4158383230362D303231302D30303030 // Ch B AxisMain parameters / Configured drive type
//         startup 13891:1 := 9A993940 // Ch B TorqueCtrl parameters / Configured channel rated current
//         startup 13891:2 := 33330B41 // Ch B TorqueCtrl parameters / Configured channel peak current
//         startup 13888:1 := EEA21643 // Ch B TorqueCtrl parameters mappable / Torque control proportional gain q
//         startup 13888:2 := 8A0E7C39 // Ch B TorqueCtrl parameters mappable / Torque control integral action time q
//         startup 13632:1 := F9F4283E // Ch B VeloCtrl parameters mappable / Velocity control proportional gain
//         startup 13632:2 := 6F12033C // Ch B VeloCtrl parameters mappable / Velocity control integral action time
//         startup 13632:3 := 00980546 // Ch B VeloCtrl parameters mappable / Bipolar velocity limit value
//         startup 14016:15 := 0100 // Ch B Motor parameters / Motor temperature sensor connection
//         startup 13635:4 := 0400 // Ch B VeloCtrl observer / Observer type
//         startup 26720:0 := 08 // Ch B Modes of operation
//         startup 13320:2 := 00 // Ch B AxisMain parameters encoder polarity / Primary encoder actual values
//         startup 13635:4 := 0400 // Ch B VeloCtrl observer / Observer type
//         startup 14095:2 := 00000000 // Ch B Secondary Feedback BiSS-C: Encoder parameter (linear) / Power supply
//         startup 14095:6 := 00 // Ch B Secondary Feedback BiSS-C: Encoder parameter (linear) / Data layout
//         startup 14095:7 := 00 // Ch B Secondary Feedback BiSS-C: Encoder parameter (linear) / Fill bit count left
//         startup 14095:8 := 00 // Ch B Secondary Feedback BiSS-C: Encoder parameter (linear) / Fill bit count right
//         startup 13320:1 := 00 // Ch B AxisMain parameters encoder polarity / Secondary encoder actual values
//       Drive 74 (AX8206-0210-0104) [AX8206-0210-0104 (2Ch. 6A servo axis, safe-motion, multi-FB)]
//         modules: Device, Device, Device, Device, Device, Device, Device, Device, Device, Device, Device (Safety), Device, Device, Device, Device, Device, Device, Device, Device, Device, Device, Device, Device, Device, Device, Device, Device, Device, Device, Device, Device, Ch A, Ch A, Ch A, Ch A, Ch A, Ch A, Ch A, Ch A, Ch A, Ch A, Ch A, Ch A, Ch A, Ch A, Ch A, Ch A, Ch A, Ch A, Ch A, Ch A, Ch A, Ch A, Ch A, Ch A, Ch A, Ch A, Ch A, Ch B, Ch B, Ch B, Ch B, Ch B, Ch B, Ch B, Ch B, Ch B, Ch B, Ch B, Ch B, Ch B, Ch B, Ch B, Ch B, Ch B, Ch B, Ch B, Ch B, Ch B, Ch B, Ch B, Ch B, Ch B, Ch B, Ch B
//         startup 12992:1 := 414D383035332D78477831 // Ch A Motor parameters / Configured motor type
//         startup 24768:0 := FEFF // Ch A Interpolation sub mode select
//         startup 13000:5 := 0200 // Ch A Motor thermal model / Reaction
//         startup 12992:12 := 0000FA44 // Ch A Motor parameters / Motor rated speed
//         startup 12992:13 := 73681F41 // Ch A Motor parameters / Motor rated torque
//         startup 24694:0 := 9D2C0000 // Ch A Motor standstill torque
//         startup 24800:0 := D007 // Ch A Positive torque/force limit value
//         startup 24801:0 := D007 // Ch A Negative torque/force limit value
//         startup 12288:6 := 4158383230362D303231302D30303030 // Ch A AxisMain parameters / Configured drive type
//         startup 12867:1 := 66669640 // Ch A TorqueCtrl parameters / Configured channel rated current
//         startup 12867:2 := 9A996141 // Ch A TorqueCtrl parameters / Configured channel peak current
//         startup 12864:1 := 0501AA42 // Ch A TorqueCtrl parameters mappable / Torque control proportional gain q
//         startup 12864:2 := 8A0E7C39 // Ch A TorqueCtrl parameters mappable / Torque control integral action time q
//         startup 12608:1 := 6832A93E // Ch A VeloCtrl parameters mappable / Velocity control proportional gain
//         startup 12608:2 := 6F12033C // Ch A VeloCtrl parameters mappable / Velocity control integral action time
//         startup 12608:3 := 00980546 // Ch A VeloCtrl parameters mappable / Bipolar velocity limit value
//         startup 12992:15 := 0100 // Ch A Motor parameters / Motor temperature sensor connection
//         startup 12611:4 := 0400 // Ch A VeloCtrl observer / Observer type
//         startup 24672:0 := 08 // Ch A Modes of operation
//         startup 12296:2 := 00 // Ch A AxisMain parameters encoder polarity / Primary encoder actual values
//         startup 12611:4 := 0400 // Ch A VeloCtrl observer / Observer type
//         startup 13071:2 := 00000000 // Ch A Secondary Feedback BiSS-C: Encoder parameter (linear) / Power supply
//         startup 13071:6 := 00 // Ch A Secondary Feedback BiSS-C: Encoder parameter (linear) / Data layout
//         startup 13071:7 := 00 // Ch A Secondary Feedback BiSS-C: Encoder parameter (linear) / Fill bit count left
//         startup 13071:8 := 00 // Ch A Secondary Feedback BiSS-C: Encoder parameter (linear) / Fill bit count right
//         startup 24672:0 := 08 // Ch A Modes of operation
//         startup 12296:1 := 00 // Ch A AxisMain parameters encoder polarity / Secondary encoder actual values
//         startup 14016:1 := 414D383035332D78477831 // Ch B Motor parameters / Configured motor type
//         startup 26816:0 := FEFF // Ch B Interpolation sub mode select
//         startup 14024:5 := 0200 // Ch B Motor thermal model / Reaction
//         startup 14016:12 := 0000FA44 // Ch B Motor parameters / Motor rated speed
//         startup 14016:13 := 73681F41 // Ch B Motor parameters / Motor rated torque
//         startup 26742:0 := 9D2C0000 // Ch B Motor standstill torque
//         startup 26848:0 := D007 // Ch B Positive torque/force limit value
//         startup 26849:0 := D007 // Ch B Negative torque/force limit value
//         startup 13312:6 := 4158383230362D303231302D30303030 // Ch B AxisMain parameters / Configured drive type
//         startup 13891:1 := 66669640 // Ch B TorqueCtrl parameters / Configured channel rated current
//         startup 13891:2 := 9A996141 // Ch B TorqueCtrl parameters / Configured channel peak current
//         startup 13888:1 := 0501AA42 // Ch B TorqueCtrl parameters mappable / Torque control proportional gain q
//         startup 13888:2 := 8A0E7C39 // Ch B TorqueCtrl parameters mappable / Torque control integral action time q
//         startup 13632:1 := 6832A93E // Ch B VeloCtrl parameters mappable / Velocity control proportional gain
//         startup 13632:2 := 6F12033C // Ch B VeloCtrl parameters mappable / Velocity control integral action time
//         startup 13632:3 := 00980546 // Ch B VeloCtrl parameters mappable / Bipolar velocity limit value
//         startup 14016:15 := 0100 // Ch B Motor parameters / Motor temperature sensor connection
//         startup 13635:4 := 0400 // Ch B VeloCtrl observer / Observer type
//         startup 26720:0 := 08 // Ch B Modes of operation
//         startup 13320:2 := 00 // Ch B AxisMain parameters encoder polarity / Primary encoder actual values
//         startup 13635:4 := 0400 // Ch B VeloCtrl observer / Observer type
//         startup 14095:2 := 00000000 // Ch B Secondary Feedback BiSS-C: Encoder parameter (linear) / Power supply
//         startup 14095:6 := 00 // Ch B Secondary Feedback BiSS-C: Encoder parameter (linear) / Data layout
//         startup 14095:7 := 00 // Ch B Secondary Feedback BiSS-C: Encoder parameter (linear) / Fill bit count left
//         startup 14095:8 := 00 // Ch B Secondary Feedback BiSS-C: Encoder parameter (linear) / Fill bit count right
//         startup 13320:1 := 00 // Ch B AxisMain parameters encoder polarity / Secondary encoder actual values
//       Term 78 (EL9011) [EL9011 End Terminal]
//   DEVICE Device 6 (NOV-DP-RAM) (disabled)
// variable links:
//   (this object) <-> Device 1 (EtherCAT)/Term 17 (EK1100)/Term 19 (EL5101)
//     Enc/Inputs/In/nDataIn1[0] <-> ENC Status compact/Counter value
//     Enc/Inputs/In/nDataIn2[0] <-> ENC Status compact/Latch value
//     Enc/Inputs/In/nState1 @bit 4 <-> ENC Status compact/Status/Counter overflow
//     Enc/Inputs/In/nState1 @bit 3 <-> ENC Status compact/Status/Counter underflow
//     Enc/Inputs/In/nState1 @bit 7 <-> ENC Status compact/Status/Extrapolation stall
//     Enc/Inputs/In/nState1 <-> ENC Status compact/Status/Latch C valid
//     Enc/Inputs/In/nState1 @bit 1 <-> ENC Status compact/Status/Latch extern valid
//     Enc/Inputs/In/nState1 @bit 6 <-> ENC Status compact/Status/Open circuit
//     Enc/Inputs/In/nState1 @bit 2 <-> ENC Status compact/Status/Set counter done
//     Enc/Inputs/In/nState1 @bit 5 <-> ENC Status compact/Status/Status of input status
//     Enc/Inputs/In/nState2 @bit 4 <-> ENC Status compact/Status/Status of extern latch
//     Enc/Inputs/In/nState2 <-> ENC Status compact/Status/Status of input A
//     Enc/Inputs/In/nState2 @bit 1 <-> ENC Status compact/Status/Status of input B
//     Enc/Inputs/In/nState2 @bit 2 <-> ENC Status compact/Status/Status of input C
//     Enc/Inputs/In/nState2 @bit 3 <-> ENC Status compact/Status/Status of input gate
//     Enc/Inputs/In/nState2 @bit 5 <-> ENC Status compact/Status/Sync error
//     Enc/Inputs/In/nState2 @bit 6 <-> ENC Status compact/Status/TxPDO State
//     Enc/Inputs/In/nState2 @bit 7 <-> ENC Status compact/Status/TxPDO Toggle
//     Enc/Inputs/In/nState4 @bit 1 <-> WcState/InputToggle
//     Enc/Inputs/In/nState4 <-> WcState/WcState
//     Enc/Outputs/Out/nCtrl1 <-> ENC Control compact/Control/Enable latch C
//     Enc/Outputs/Out/nCtrl1 @bit 3 <-> ENC Control compact/Control/Enable latch extern on negative edge
//     Enc/Outputs/Out/nCtrl1 @bit 1 <-> ENC Control compact/Control/Enable latch extern on positive edge
//     Enc/Outputs/Out/nCtrl1 @bit 2 <-> ENC Control compact/Control/Set counter
//     Enc/Outputs/Out/nDataOut1[0] <-> ENC Control compact/Set counter value
//   (this object) <-> Device 1 (EtherCAT)/Term 22 (EK1100)/Term 23 (EL7047)
//     Drive/Inputs/In/nState1 @bit 3 <-> STM Status/Status/Error
//     Drive/Inputs/In/nState1 @bit 7 <-> STM Status/Status/Motor stall
//     Drive/Inputs/In/nState1 @bit 5 <-> STM Status/Status/Moving negative
//     Drive/Inputs/In/nState1 @bit 4 <-> STM Status/Status/Moving positive
//     Drive/Inputs/In/nState1 @bit 1 <-> STM Status/Status/Ready
//     Drive/Inputs/In/nState1 <-> STM Status/Status/Ready to enable
//     Drive/Inputs/In/nState1 @bit 6 <-> STM Status/Status/Torque reduced
//     Drive/Inputs/In/nState1 @bit 2 <-> STM Status/Status/Warning
//     Drive/Inputs/In/nState2 @bit 3 <-> STM Status/Status/Digital input 1
//     Drive/Inputs/In/nState2 @bit 4 <-> STM Status/Status/Digital input 2
//     Drive/Inputs/In/nState2 @bit 5 <-> STM Status/Status/Sync error
//     Drive/Inputs/In/nState2 @bit 7 <-> STM Status/Status/TxPDO Toggle
//     Drive/Inputs/In/nState4 @bit 1 <-> WcState/InputToggle
//     Drive/Inputs/In/nState4 <-> WcState/WcState
//     Drive/Outputs/Out/nCtrl1 <-> STM Control/Control/Enable
//     Drive/Outputs/Out/nCtrl1 @bit 2 <-> STM Control/Control/Reduce torque
//     Drive/Outputs/Out/nCtrl1 @bit 1 <-> STM Control/Control/Reset
//     Drive/Outputs/Out/nCtrl2 @bit 3 <-> STM Control/Control/Digital output 1
//     Drive/Outputs/Out/nDataOut2[0] <-> STM Velocity/Velocity
//   (this object) <-> Device 1 (EtherCAT)/Term 17 (EK1100)/Term 18 (EL5101)
//     Enc/Inputs/In/nDataIn1[0] <-> ENC Status compact/Counter value
//     Enc/Inputs/In/nDataIn2[0] <-> ENC Status compact/Latch value
//     Enc/Inputs/In/nState1 @bit 4 <-> ENC Status compact/Status/Counter overflow
//     Enc/Inputs/In/nState1 @bit 3 <-> ENC Status compact/Status/Counter underflow
//     Enc/Inputs/In/nState1 @bit 7 <-> ENC Status compact/Status/Extrapolation stall
//     Enc/Inputs/In/nState1 <-> ENC Status compact/Status/Latch C valid
//     Enc/Inputs/In/nState1 @bit 1 <-> ENC Status compact/Status/Latch extern valid
//     Enc/Inputs/In/nState1 @bit 6 <-> ENC Status compact/Status/Open circuit
//     Enc/Inputs/In/nState1 @bit 2 <-> ENC Status compact/Status/Set counter done
//     Enc/Inputs/In/nState1 @bit 5 <-> ENC Status compact/Status/Status of input status
//     Enc/Inputs/In/nState2 @bit 4 <-> ENC Status compact/Status/Status of extern latch
//     Enc/Inputs/In/nState2 <-> ENC Status compact/Status/Status of input A
//     Enc/Inputs/In/nState2 @bit 1 <-> ENC Status compact/Status/Status of input B
//     Enc/Inputs/In/nState2 @bit 2 <-> ENC Status compact/Status/Status of input C
//     Enc/Inputs/In/nState2 @bit 3 <-> ENC Status compact/Status/Status of input gate
//     Enc/Inputs/In/nState2 @bit 5 <-> ENC Status compact/Status/Sync error
//     Enc/Inputs/In/nState2 @bit 6 <-> ENC Status compact/Status/TxPDO State
//     Enc/Inputs/In/nState2 @bit 7 <-> ENC Status compact/Status/TxPDO Toggle
//     Enc/Inputs/In/nState4 @bit 1 <-> WcState/InputToggle
//     Enc/Inputs/In/nState4 <-> WcState/WcState
//     Enc/Outputs/Out/nCtrl1 <-> ENC Control compact/Control/Enable latch C
//     Enc/Outputs/Out/nCtrl1 @bit 3 <-> ENC Control compact/Control/Enable latch extern on negative edge
//     Enc/Outputs/Out/nCtrl1 @bit 1 <-> ENC Control compact/Control/Enable latch extern on positive edge
//     Enc/Outputs/Out/nCtrl1 @bit 2 <-> ENC Control compact/Control/Set counter
//     Enc/Outputs/Out/nDataOut1[0] <-> ENC Control compact/Set counter value
//   (this object) <-> Device 1 (EtherCAT)/Term 22 (EK1100)/Term 24 (EL7047)
//     Drive/Inputs/In/nState1 @bit 3 <-> STM Status/Status/Error
//     Drive/Inputs/In/nState1 @bit 7 <-> STM Status/Status/Motor stall
//     Drive/Inputs/In/nState1 @bit 5 <-> STM Status/Status/Moving negative
//     Drive/Inputs/In/nState1 @bit 4 <-> STM Status/Status/Moving positive
//     Drive/Inputs/In/nState1 @bit 1 <-> STM Status/Status/Ready
//     Drive/Inputs/In/nState1 <-> STM Status/Status/Ready to enable
//     Drive/Inputs/In/nState1 @bit 6 <-> STM Status/Status/Torque reduced
//     Drive/Inputs/In/nState1 @bit 2 <-> STM Status/Status/Warning
//     Drive/Inputs/In/nState2 @bit 3 <-> STM Status/Status/Digital input 1
//     Drive/Inputs/In/nState2 @bit 4 <-> STM Status/Status/Digital input 2
//     Drive/Inputs/In/nState2 @bit 5 <-> STM Status/Status/Sync error
//     Drive/Inputs/In/nState2 @bit 7 <-> STM Status/Status/TxPDO Toggle
//     Drive/Inputs/In/nState4 @bit 1 <-> WcState/InputToggle
//     Drive/Inputs/In/nState4 <-> WcState/WcState
//     Drive/Outputs/Out/nCtrl1 <-> STM Control/Control/Enable
//     Drive/Outputs/Out/nCtrl1 @bit 2 <-> STM Control/Control/Reduce torque
//     Drive/Outputs/Out/nCtrl1 @bit 1 <-> STM Control/Control/Reset
//     Drive/Outputs/Out/nCtrl2 @bit 3 <-> STM Control/Control/Digital output 1
//     Drive/Outputs/Out/nDataOut2[0] <-> STM Velocity/Velocity
//   (this object) <-> Device 1 (EtherCAT)/Term 17 (EK1100)/Term 21 (EL5101)
//     Enc/Inputs/In/nDataIn1[0] <-> ENC Status compact/Counter value
//     Enc/Inputs/In/nDataIn2[0] <-> ENC Status compact/Latch value
//     Enc/Inputs/In/nState1 @bit 4 <-> ENC Status compact/Status/Counter overflow
//     Enc/Inputs/In/nState1 @bit 3 <-> ENC Status compact/Status/Counter underflow
//     Enc/Inputs/In/nState1 @bit 7 <-> ENC Status compact/Status/Extrapolation stall
//     Enc/Inputs/In/nState1 <-> ENC Status compact/Status/Latch C valid
//     Enc/Inputs/In/nState1 @bit 1 <-> ENC Status compact/Status/Latch extern valid
//     Enc/Inputs/In/nState1 @bit 6 <-> ENC Status compact/Status/Open circuit
//     Enc/Inputs/In/nState1 @bit 2 <-> ENC Status compact/Status/Set counter done
//     Enc/Inputs/In/nState1 @bit 5 <-> ENC Status compact/Status/Status of input status
//     Enc/Inputs/In/nState2 @bit 4 <-> ENC Status compact/Status/Status of extern latch
//     Enc/Inputs/In/nState2 <-> ENC Status compact/Status/Status of input A
//     Enc/Inputs/In/nState2 @bit 1 <-> ENC Status compact/Status/Status of input B
//     Enc/Inputs/In/nState2 @bit 2 <-> ENC Status compact/Status/Status of input C
//     Enc/Inputs/In/nState2 @bit 3 <-> ENC Status compact/Status/Status of input gate
//     Enc/Inputs/In/nState2 @bit 5 <-> ENC Status compact/Status/Sync error
//     Enc/Inputs/In/nState2 @bit 6 <-> ENC Status compact/Status/TxPDO State
//     Enc/Inputs/In/nState2 @bit 7 <-> ENC Status compact/Status/TxPDO Toggle
//     Enc/Inputs/In/nState4 @bit 1 <-> WcState/InputToggle
//     Enc/Inputs/In/nState4 <-> WcState/WcState
//     Enc/Outputs/Out/nCtrl1 <-> ENC Control compact/Control/Enable latch C
//     Enc/Outputs/Out/nCtrl1 @bit 3 <-> ENC Control compact/Control/Enable latch extern on negative edge
//     Enc/Outputs/Out/nCtrl1 @bit 1 <-> ENC Control compact/Control/Enable latch extern on positive edge
//     Enc/Outputs/Out/nCtrl1 @bit 2 <-> ENC Control compact/Control/Set counter
//     Enc/Outputs/Out/nDataOut1[0] <-> ENC Control compact/Set counter value
//   (this object) <-> Device 1 (EtherCAT)/Term 22 (EK1100)/Term 25 (EL7047)
//     Drive/Inputs/In/nState1 @bit 3 <-> STM Status/Status/Error
//     Drive/Inputs/In/nState1 @bit 7 <-> STM Status/Status/Motor stall
//     Drive/Inputs/In/nState1 @bit 5 <-> STM Status/Status/Moving negative
//     Drive/Inputs/In/nState1 @bit 4 <-> STM Status/Status/Moving positive
//     Drive/Inputs/In/nState1 @bit 1 <-> STM Status/Status/Ready
//     Drive/Inputs/In/nState1 <-> STM Status/Status/Ready to enable
//     Drive/Inputs/In/nState1 @bit 6 <-> STM Status/Status/Torque reduced
//     Drive/Inputs/In/nState1 @bit 2 <-> STM Status/Status/Warning
//     Drive/Inputs/In/nState2 @bit 3 <-> STM Status/Status/Digital input 1
//     Drive/Inputs/In/nState2 @bit 4 <-> STM Status/Status/Digital input 2
//     Drive/Inputs/In/nState2 @bit 5 <-> STM Status/Status/Sync error
//     Drive/Inputs/In/nState2 @bit 7 <-> STM Status/Status/TxPDO Toggle
//     Drive/Inputs/In/nState4 @bit 1 <-> WcState/InputToggle
//     Drive/Inputs/In/nState4 <-> WcState/WcState
//     Drive/Outputs/Out/nCtrl1 <-> STM Control/Control/Enable
//     Drive/Outputs/Out/nCtrl1 @bit 2 <-> STM Control/Control/Reduce torque
//     Drive/Outputs/Out/nCtrl1 @bit 1 <-> STM Control/Control/Reset
//     Drive/Outputs/Out/nCtrl2 @bit 3 <-> STM Control/Control/Digital output 1
//     Drive/Outputs/Out/nDataOut2[0] <-> STM Velocity/Velocity
//   (this object) <-> Device 1 (EtherCAT)/Term 17 (EK1100)/Term 20 (EL5101)
//     Enc/Inputs/In/nDataIn1[0] <-> ENC Status compact/Counter value
//     Enc/Inputs/In/nDataIn2[0] <-> ENC Status compact/Latch value
//     Enc/Inputs/In/nState1 @bit 4 <-> ENC Status compact/Status/Counter overflow
//     Enc/Inputs/In/nState1 @bit 3 <-> ENC Status compact/Status/Counter underflow
//     Enc/Inputs/In/nState1 @bit 7 <-> ENC Status compact/Status/Extrapolation stall
//     Enc/Inputs/In/nState1 <-> ENC Status compact/Status/Latch C valid
//     Enc/Inputs/In/nState1 @bit 1 <-> ENC Status compact/Status/Latch extern valid
//     Enc/Inputs/In/nState1 @bit 6 <-> ENC Status compact/Status/Open circuit
//     Enc/Inputs/In/nState1 @bit 2 <-> ENC Status compact/Status/Set counter done
//     Enc/Inputs/In/nState1 @bit 5 <-> ENC Status compact/Status/Status of input status
//     Enc/Inputs/In/nState2 @bit 4 <-> ENC Status compact/Status/Status of extern latch
//     Enc/Inputs/In/nState2 <-> ENC Status compact/Status/Status of input A
//     Enc/Inputs/In/nState2 @bit 1 <-> ENC Status compact/Status/Status of input B
//     Enc/Inputs/In/nState2 @bit 2 <-> ENC Status compact/Status/Status of input C
//     Enc/Inputs/In/nState2 @bit 3 <-> ENC Status compact/Status/Status of input gate
//     Enc/Inputs/In/nState2 @bit 5 <-> ENC Status compact/Status/Sync error
//     Enc/Inputs/In/nState2 @bit 6 <-> ENC Status compact/Status/TxPDO State
//     Enc/Inputs/In/nState2 @bit 7 <-> ENC Status compact/Status/TxPDO Toggle
//     Enc/Inputs/In/nState4 @bit 1 <-> WcState/InputToggle
//     Enc/Inputs/In/nState4 <-> WcState/WcState
//     Enc/Outputs/Out/nCtrl1 <-> ENC Control compact/Control/Enable latch C
//     Enc/Outputs/Out/nCtrl1 @bit 3 <-> ENC Control compact/Control/Enable latch extern on negative edge
//     Enc/Outputs/Out/nCtrl1 @bit 1 <-> ENC Control compact/Control/Enable latch extern on positive edge
//     Enc/Outputs/Out/nCtrl1 @bit 2 <-> ENC Control compact/Control/Set counter
//     Enc/Outputs/Out/nDataOut1[0] <-> ENC Control compact/Set counter value
//   (this object) <-> Device 1 (EtherCAT)/Term 22 (EK1100)/Term 26 (EL7047)
//     Drive/Inputs/In/nState1 @bit 3 <-> STM Status/Status/Error
//     Drive/Inputs/In/nState1 @bit 7 <-> STM Status/Status/Motor stall
//     Drive/Inputs/In/nState1 @bit 5 <-> STM Status/Status/Moving negative
//     Drive/Inputs/In/nState1 @bit 4 <-> STM Status/Status/Moving positive
//     Drive/Inputs/In/nState1 @bit 1 <-> STM Status/Status/Ready
//     Drive/Inputs/In/nState1 <-> STM Status/Status/Ready to enable
//     Drive/Inputs/In/nState1 @bit 6 <-> STM Status/Status/Torque reduced
//     Drive/Inputs/In/nState1 @bit 2 <-> STM Status/Status/Warning
//     Drive/Inputs/In/nState2 @bit 3 <-> STM Status/Status/Digital input 1
//     Drive/Inputs/In/nState2 @bit 4 <-> STM Status/Status/Digital input 2
//     Drive/Inputs/In/nState2 @bit 5 <-> STM Status/Status/Sync error
//     Drive/Inputs/In/nState2 @bit 7 <-> STM Status/Status/TxPDO Toggle
//     Drive/Inputs/In/nState4 @bit 1 <-> WcState/InputToggle
//     Drive/Inputs/In/nState4 <-> WcState/WcState
//     Drive/Outputs/Out/nCtrl1 <-> STM Control/Control/Enable
//     Drive/Outputs/Out/nCtrl1 @bit 2 <-> STM Control/Control/Reduce torque
//     Drive/Outputs/Out/nCtrl1 @bit 1 <-> STM Control/Control/Reset
//     Drive/Outputs/Out/nCtrl2 @bit 3 <-> STM Control/Control/Digital output 1
//     Drive/Outputs/Out/nDataOut2[0] <-> STM Velocity/Velocity
//   (this object) <-> Device 1 (EtherCAT)/Term 70 (AX8640-0000-0103)/Drive 71 (AX8206-0210-0104)
//     Drive/Inputs/In/nDataIn1 <-> Ch A/Ch A PositionControl Inputs/Ch A Following error actual value
//     Drive/Inputs/In/nDataIn3[0] <-> Ch A/Ch A TorqueControl Inputs/Ch A Torque/force actual value
//     Drive/Inputs/In/nDcOutputTime <-> InfoData/DcOutputShift
//     Drive/Inputs/In/nState1 <-> Ch A/Ch A AxisMain Inputs/Ch A Statusword
//     Drive/Inputs/In/nState2 <-> Ch A/Ch A AxisMain Inputs/Ch A Statusword @bit 8
//     Drive/Inputs/In/nState4 @bit 1 <-> WcState/InputToggle0
//     Drive/Inputs/In/nState4 <-> WcState/WcState0
//     Drive/Inputs/In/nState5 <-> Ch A/Ch A AxisMain Inputs/Ch A Modes of operation display
//     Drive/Outputs/Out/nCtrl1 <-> Ch A/Ch A AxisMain Outputs/Ch A Controlword
//     Drive/Outputs/Out/nCtrl2 <-> Ch A/Ch A AxisMain Outputs/Ch A Controlword @bit 8
//     Drive/Outputs/Out/nCtrl5 <-> Ch A/Ch A AxisMain Outputs/Ch A Modes of operation
//     Drive/Outputs/Out/nDataOut1 <-> Ch A/Ch A Interpolator Outputs/Ch A Target position
//     Drive/Outputs/Out/nDataOut2 <-> Ch A/Ch A Interpolator Outputs/Ch A Target velocity
//     Drive/Outputs/Out/nDataOut4[0] <-> Ch A/Ch A TorqueControl Outputs/Ch A Target torque/force
//     Enc/Inputs/In/nDataIn1 <-> Ch A/Ch A AxisMain Inputs/Ch A Position actual value
//     Enc/Inputs/In/nDataIn4 @bit 5 <-> Ch A/Ch A AxisMain Inputs/Position actual value invalid
//     Enc/Inputs/In/nDataIn6 @bit 1 <-> WcState/InputToggle0
//     Enc/Inputs/In/nDataIn6 <-> WcState/WcState0
//     Enc/Inputs/In/nDcInputTime <-> InfoData/DcInputShift
//     Drive/Inputs/In/nDataIn1 <-> Ch B/Ch B PositionControl Inputs/Ch B Following error actual value
//     Drive/Inputs/In/nDataIn3[0] <-> Ch B/Ch B TorqueControl Inputs/Ch B Torque/force actual value
//     Drive/Inputs/In/nState1 <-> Ch B/Ch B AxisMain Inputs/Ch B Statusword
//     Drive/Inputs/In/nState2 <-> Ch B/Ch B AxisMain Inputs/Ch B Statusword @bit 8
//     Drive/Outputs/Out/nCtrl1 <-> Ch B/Ch B AxisMain Outputs/Ch B Controlword
//     Drive/Outputs/Out/nCtrl2 <-> Ch B/Ch B AxisMain Outputs/Ch B Controlword @bit 8
//     Drive/Outputs/Out/nDataOut1 <-> Ch B/Ch B Interpolator Outputs/Ch B Target position
//     Drive/Outputs/Out/nDataOut2 <-> Ch B/Ch B Interpolator Outputs/Ch B Target velocity
//     Enc/Inputs/In/nDataIn1 <-> Ch B/Ch B AxisMain Inputs/1st additional position actual value
//     Enc/Inputs/In/nState2 @bit 5 <-> Ch B/Ch B AxisMain Inputs/1st Additional position actual value invalid
//     Enc/Inputs/In/nState4 @bit 1 <-> WcState/InputToggle0
//     Enc/Inputs/In/nState4 <-> WcState/WcState0
//     Enc/Inputs/In/nDataIn1 <-> Ch A/Ch A AxisMain Inputs/1st additional position actual value
//     Term 27 (EK1100)/EL6910-(04)/ConnectionInputs/Message_5 TxPDO <-> Device (Safety)/FSoE Slave Connection 1 Master Message/Message_1
//     Term 27 (EK1100)/EL6910-(04)/ConnectionOutputs/Message_5 RxPDO <-> Device (Safety)/FSoE Slave Connection 1 Slave Message/Message_1
//     Term 70 (AX8640-0000-0103)/PSM Controlword for axis/Controlword for axis <-> Device/DeviceMain Outputs/Power supply controlword
//   (this object) <-> Device 1 (EtherCAT)/Term 70 (AX8640-0000-0103)/Drive 74 (AX8206-0210-0104)
//     Drive/Inputs/In/nDataIn1 <-> Ch A/Ch A PositionControl Inputs/Ch A Following error actual value
//     Drive/Inputs/In/nDataIn3[0] <-> Ch A/Ch A TorqueControl Inputs/Ch A Torque/force actual value
//     Drive/Inputs/In/nDcOutputTime <-> InfoData/DcOutputShift
//     Drive/Inputs/In/nState1 <-> Ch A/Ch A AxisMain Inputs/Ch A Statusword
//     Drive/Inputs/In/nState2 <-> Ch A/Ch A AxisMain Inputs/Ch A Statusword @bit 8
//     Drive/Inputs/In/nState4 @bit 1 <-> WcState/InputToggle0
//     Drive/Inputs/In/nState4 <-> WcState/WcState0
//     Drive/Outputs/Out/nCtrl1 <-> Ch A/Ch A AxisMain Outputs/Ch A Controlword
//     Drive/Outputs/Out/nCtrl2 <-> Ch A/Ch A AxisMain Outputs/Ch A Controlword @bit 8
//     Drive/Outputs/Out/nDataOut1 <-> Ch A/Ch A Interpolator Outputs/Ch A Target position
//     Drive/Outputs/Out/nDataOut2 <-> Ch A/Ch A Interpolator Outputs/Ch A Target velocity
//     Enc/Inputs/In/nDataIn1 <-> Ch A/Ch A AxisMain Inputs/1st additional position actual value
//     Enc/Inputs/In/nDcInputTime <-> InfoData/DcInputShift
//     Enc/Inputs/In/nState2 @bit 5 <-> Ch A/Ch A AxisMain Inputs/1st Additional position actual value invalid
//     Enc/Inputs/In/nState4 @bit 1 <-> WcState/InputToggle0
//     Enc/Inputs/In/nState4 <-> WcState/WcState0
//     Drive/Inputs/In/nDataIn1 <-> Ch B/Ch B PositionControl Inputs/Ch B Following error actual value
//     Drive/Inputs/In/nDataIn3[0] <-> Ch B/Ch B TorqueControl Inputs/Ch B Torque/force actual value
//     Drive/Inputs/In/nState1 <-> Ch B/Ch B AxisMain Inputs/Ch B Statusword
//     Drive/Inputs/In/nState2 <-> Ch B/Ch B AxisMain Inputs/Ch B Statusword @bit 8
//     Drive/Outputs/Out/nCtrl1 <-> Ch B/Ch B AxisMain Outputs/Ch B Controlword
//     Drive/Outputs/Out/nCtrl2 <-> Ch B/Ch B AxisMain Outputs/Ch B Controlword @bit 8
//     Drive/Outputs/Out/nDataOut1 <-> Ch B/Ch B Interpolator Outputs/Ch B Target position
//     Drive/Outputs/Out/nDataOut2 <-> Ch B/Ch B Interpolator Outputs/Ch B Target velocity
//     Enc/Inputs/In/nDataIn1 <-> Ch B/Ch B AxisMain Inputs/1st additional position actual value
//     Enc/Inputs/In/nState2 @bit 5 <-> Ch B/Ch B AxisMain Inputs/1st Additional position actual value invalid
//     Term 27 (EK1100)/EL6910-(04)/ConnectionInputs/Message_6 TxPDO <-> Device (Safety)/FSoE Slave Connection 1 Master Message/Message_1
//     Term 27 (EK1100)/EL6910-(04)/ConnectionOutputs/Message_6 RxPDO <-> Device (Safety)/FSoE Slave Connection 1 Slave Message/Message_1
//     Term 70 (AX8640-0000-0103)/PSM Controlword for axis/Controlword for axis <-> Device/DeviceMain Outputs/Power supply controlword
//   (this object) <-> Device 1 (EtherCAT)/Term 27 (EK1100)/EL1904-(06)
//     Term 27 (EK1100)/EL6910-(04)/ConnectionInputs/Message_10 TxPDO <-> Module 1 (FSOES)/RxPDO/FSOE
//     Term 27 (EK1100)/EL6910-(04)/ConnectionOutputs/Message_10 RxPDO <-> Module 1 (FSOES)/TxPDO/FSOE
//   (this object) <-> Device 1 (EtherCAT)/Term 27 (EK1100)/EL1904-(07)
//     Term 27 (EK1100)/EL6910-(04)/ConnectionInputs/Message_11 TxPDO <-> Module 1 (FSOES)/RxPDO/FSOE
//     Term 27 (EK1100)/EL6910-(04)/ConnectionOutputs/Message_11 RxPDO <-> Module 1 (FSOES)/TxPDO/FSOE
//   (this object) <-> Device 1 (EtherCAT)/Term 27 (EK1100)/EL1904-(08)
//     Term 27 (EK1100)/EL6910-(04)/ConnectionInputs/Message_7 TxPDO <-> Module 1 (FSOES)/RxPDO/FSOE
//     Term 27 (EK1100)/EL6910-(04)/ConnectionOutputs/Message_7 RxPDO <-> Module 1 (FSOES)/TxPDO/FSOE
//   (this object) <-> Device 1 (EtherCAT)/Term 27 (EK1100)/EL1904-(09)
//     Term 27 (EK1100)/EL6910-(04)/ConnectionInputs/Message_12 TxPDO <-> Module 1 (FSOES)/RxPDO/FSOE
//     Term 27 (EK1100)/EL6910-(04)/ConnectionOutputs/Message_12 RxPDO <-> Module 1 (FSOES)/TxPDO/FSOE
//   (this object) <-> Device 1 (EtherCAT)/Term 27 (EK1100)/EL1904-(10)
//     Term 27 (EK1100)/EL6910-(04)/ConnectionInputs/Message_13 TxPDO <-> Module 1 (FSOES)/RxPDO/FSOE
//     Term 27 (EK1100)/EL6910-(04)/ConnectionOutputs/Message_13 RxPDO <-> Module 1 (FSOES)/TxPDO/FSOE
//   (this object) <-> Device 1 (EtherCAT)/Term 27 (EK1100)/EL1904-(11)
//     Term 27 (EK1100)/EL6910-(04)/ConnectionInputs/Message_14 TxPDO <-> Module 1 (FSOES)/RxPDO/FSOE
//     Term 27 (EK1100)/EL6910-(04)/ConnectionOutputs/Message_14 RxPDO <-> Module 1 (FSOES)/TxPDO/FSOE
//   (this object) <-> Device 1 (EtherCAT)/Term 27 (EK1100)/EL1904-(12)
//     Term 27 (EK1100)/EL6910-(04)/ConnectionInputs/Message_17 TxPDO <-> Module 1 (FSOES)/RxPDO/FSOE
//     Term 27 (EK1100)/EL6910-(04)/ConnectionOutputs/Message_17 RxPDO <-> Module 1 (FSOES)/TxPDO/FSOE
//   (this object) <-> Device 1 (EtherCAT)/Term 27 (EK1100)/EL1904-(13)
//     Term 27 (EK1100)/EL6910-(04)/ConnectionInputs/Message_18 TxPDO <-> Module 1 (FSOES)/RxPDO/FSOE
//     Term 27 (EK1100)/EL6910-(04)/ConnectionOutputs/Message_18 RxPDO <-> Module 1 (FSOES)/TxPDO/FSOE
//   (this object) <-> Device 1 (EtherCAT)/Term 27 (EK1100)/EL2904-(06)
//     Term 27 (EK1100)/EL6910-(04)/ConnectionInputs/Message_8 TxPDO <-> Module 1 (FSOES)/RxPDO/FSOE
//     Term 27 (EK1100)/EL6910-(04)/ConnectionOutputs/Message_8 RxPDO <-> Module 1 (FSOES)/TxPDO/FSOE
//   (this object) <-> Device 1 (EtherCAT)/Term 27 (EK1100)/EL2904-(08)
//     Term 27 (EK1100)/EL6910-(04)/ConnectionInputs/Message_15 TxPDO <-> Module 1 (FSOES)/RxPDO/FSOE
//     Term 27 (EK1100)/EL6910-(04)/ConnectionOutputs/Message_15 RxPDO <-> Module 1 (FSOES)/TxPDO/FSOE
//   (this object) <-> Device 1 (EtherCAT)/Term 27 (EK1100)/EL2904-(09)
//     Term 27 (EK1100)/EL6910-(04)/ConnectionInputs/Message_16 TxPDO <-> Module 1 (FSOES)/RxPDO/FSOE
//     Term 27 (EK1100)/EL6910-(04)/ConnectionOutputs/Message_16 RxPDO <-> Module 1 (FSOES)/TxPDO/FSOE
//   (this object) <-> Device 1 (EtherCAT)/Term 27 (EK1100)/EL2912-(07)
//     Term 27 (EK1100)/EL6910-(04)/ConnectionInputs/Message_9 TxPDO <-> Module 1 (FSOE)/FSoE Outputs/FSOE
//     Term 27 (EK1100)/EL6910-(04)/ConnectionOutputs/Message_9 RxPDO <-> Module 1 (FSOE)/FSoE Inputs/FSOE
//   (this object) <-> Device 1 (EtherCAT)/Term 27 (EK1100)/EL6910-(04)
//     Term 27 (EK1100)/EL1904-(06)/Module 1 (FSOES)/RxPDO/FSOE <-> ConnectionInputs/Message_10 TxPDO
//     Term 27 (EK1100)/EL1904-(07)/Module 1 (FSOES)/RxPDO/FSOE <-> ConnectionInputs/Message_11 TxPDO
//     Term 27 (EK1100)/EL1904-(08)/Module 1 (FSOES)/RxPDO/FSOE <-> ConnectionInputs/Message_7 TxPDO
//     Term 27 (EK1100)/EL1904-(09)/Module 1 (FSOES)/RxPDO/FSOE <-> ConnectionInputs/Message_12 TxPDO
//     Term 27 (EK1100)/EL1904-(10)/Module 1 (FSOES)/RxPDO/FSOE <-> ConnectionInputs/Message_13 TxPDO
//     Term 27 (EK1100)/EL1904-(11)/Module 1 (FSOES)/RxPDO/FSOE <-> ConnectionInputs/Message_14 TxPDO
//     Term 27 (EK1100)/EL1904-(12)/Module 1 (FSOES)/RxPDO/FSOE <-> ConnectionInputs/Message_17 TxPDO
//     Term 27 (EK1100)/EL1904-(13)/Module 1 (FSOES)/RxPDO/FSOE <-> ConnectionInputs/Message_18 TxPDO
//     Term 27 (EK1100)/EL2904-(06)/Module 1 (FSOES)/RxPDO/FSOE <-> ConnectionInputs/Message_8 TxPDO
//     Term 27 (EK1100)/EL2904-(08)/Module 1 (FSOES)/RxPDO/FSOE <-> ConnectionInputs/Message_15 TxPDO
//     Term 27 (EK1100)/EL2904-(09)/Module 1 (FSOES)/RxPDO/FSOE <-> ConnectionInputs/Message_16 TxPDO
//     Term 27 (EK1100)/EL1904-(06)/Module 1 (FSOES)/TxPDO/FSOE <-> ConnectionOutputs/Message_10 RxPDO
//     Term 27 (EK1100)/EL1904-(07)/Module 1 (FSOES)/TxPDO/FSOE <-> ConnectionOutputs/Message_11 RxPDO
//     Term 27 (EK1100)/EL1904-(08)/Module 1 (FSOES)/TxPDO/FSOE <-> ConnectionOutputs/Message_7 RxPDO
//     Term 27 (EK1100)/EL1904-(09)/Module 1 (FSOES)/TxPDO/FSOE <-> ConnectionOutputs/Message_12 RxPDO
//     Term 27 (EK1100)/EL1904-(10)/Module 1 (FSOES)/TxPDO/FSOE <-> ConnectionOutputs/Message_13 RxPDO
//     Term 27 (EK1100)/EL1904-(11)/Module 1 (FSOES)/TxPDO/FSOE <-> ConnectionOutputs/Message_14 RxPDO
//     Term 27 (EK1100)/EL1904-(12)/Module 1 (FSOES)/TxPDO/FSOE <-> ConnectionOutputs/Message_17 RxPDO
//     Term 27 (EK1100)/EL1904-(13)/Module 1 (FSOES)/TxPDO/FSOE <-> ConnectionOutputs/Message_18 RxPDO
//     Term 27 (EK1100)/EL2904-(06)/Module 1 (FSOES)/TxPDO/FSOE <-> ConnectionOutputs/Message_8 RxPDO
//     Term 27 (EK1100)/EL2904-(08)/Module 1 (FSOES)/TxPDO/FSOE <-> ConnectionOutputs/Message_15 RxPDO
//     Term 27 (EK1100)/EL2904-(09)/Module 1 (FSOES)/TxPDO/FSOE <-> ConnectionOutputs/Message_16 RxPDO
//     Term 27 (EK1100)/EL2912-(07)/Module 1 (FSOE)/FSoE Inputs/FSOE <-> ConnectionOutputs/Message_9 RxPDO
//     Term 27 (EK1100)/EL2912-(07)/Module 1 (FSOE)/FSoE Outputs/FSOE <-> ConnectionInputs/Message_9 TxPDO
//     Term 70 (AX8640-0000-0103)/Drive 71 (AX8206-0210-0104)/Device (Safety)/FSoE Slave Connection 1 Master Message/Message_1 <-> ConnectionInputs/Message_5 TxPDO
//     Term 70 (AX8640-0000-0103)/Drive 74 (AX8206-0210-0104)/Device (Safety)/FSoE Slave Connection 1 Master Message/Message_1 <-> ConnectionInputs/Message_6 TxPDO
//     Term 70 (AX8640-0000-0103)/Drive 71 (AX8206-0210-0104)/Device (Safety)/FSoE Slave Connection 1 Slave Message/Message_1 <-> ConnectionOutputs/Message_5 RxPDO
//     Term 70 (AX8640-0000-0103)/Drive 74 (AX8206-0210-0104)/Device (Safety)/FSoE Slave Connection 1 Slave Message/Message_1 <-> ConnectionOutputs/Message_6 RxPDO
//   (this object) <-> Device 1 (EtherCAT)/Term 70 (AX8640-0000-0103)
//     Term 70 (AX8640-0000-0103)/Drive 71 (AX8206-0210-0104)/Device/DeviceMain Outputs/Power supply controlword <-> PSM Controlword for axis/Controlword for axis
//     Term 70 (AX8640-0000-0103)/Drive 74 (AX8206-0210-0104)/Device/DeviceMain Outputs/Power supply controlword <-> PSM Controlword for axis/Controlword for axis
//   tc_project_app Instance <-> Device 1 (EtherCAT)/Term 1 (EK1200)/EL10088-(03)
//     PlcTask Inputs/GVL.astAxes[1].stInputs.bLimitBwd <-> Channel 2/M1_Neg_Lim
//     PlcTask Inputs/GVL.astAxes[2].stInputs.bLimitBwd <-> Channel 3/M2_Neg_Lim
//     PlcTask Inputs/GVL.astAxes[3].stInputs.bLimitBwd <-> Channel 6/M3_Neg_Lim
//     PlcTask Inputs/GVL.astAxes[4].stInputs.bLimitBwd <-> Channel 7/M4_Neg_Lim
//     PlcTask Inputs/GVL.astAxes[1].stInputs.bLimitFwd <-> Channel 1/M1_Pos_Lim
//     PlcTask Inputs/GVL.astAxes[2].stInputs.bLimitFwd <-> Channel 4/M2_Pos_Lim
//     PlcTask Inputs/GVL.astAxes[3].stInputs.bLimitFwd <-> Channel 5/M3_Pos_Lim
//     PlcTask Inputs/GVL.astAxes[4].stInputs.bLimitFwd <-> Channel 8/M4_Pos_Lim
//   tc_project_app Instance <-> Device 1 (EtherCAT)/Term 1 (EK1200)/EL2008-(02)
//     PlcTask Outputs/Horizontal_Translation.bBwdLimitPower <-> Channel 2/Horizontal Bwd Limit Out
//     PlcTask Outputs/Horizontal_Translation.bFwdLimitPower <-> Channel 1/Horizontal Fwd Limit Out
//     PlcTask Outputs/Rotation.bBwdLimitPower <-> Channel 8/Rotation Bwd Limit Out
//     PlcTask Outputs/Rotation.bFwdLimitPower <-> Channel 7/Rotation Fwd Limit Out
//     PlcTask Outputs/Vertical_Translation_Y1.bBwdLimitPower <-> Channel 4/Vertical Z1 Bwd Limit Out
//     PlcTask Outputs/Vertical_Translation_Y2.bBwdLimitPower <-> Channel 6/Vertical Z2 Bwd Limit Out
//     PlcTask Outputs/Vertical_Translation_Y1.bFwdLimitPower <-> Channel 3/Vertical Z1 Fwd Limit Out
//     PlcTask Outputs/Vertical_Translation_Y2.bFwdLimitPower <-> Channel 5/Vertical Z2 Fwd Limit Out
//   tc_project_app Instance <-> Device 1 (EtherCAT)/Term 1 (EK1200)/EL2008-(03)
//     PlcTask Outputs/Slit_3.EastWestPowerOutput <-> Channel 2/M3_M4_Limits
//     PlcTask Outputs/Slit_3.NorthSouthPowerOutput <-> Channel 1/M1_M2_Limits
//   tc_project_app Instance <-> Device 1 (EtherCAT)/Term 1 (EK1200)/Term 50 (EL3152)
//     PlcTask Inputs/Inclinometer.INC_VAL <-> AI Standard Channel 1/Value
//   tc_project_app Instance <-> Device 1 (EtherCAT)/Term 1 (EK1200)/Term 9 (EL1008)
//     PlcTask Inputs/GVL.astAxes[5].stInputs.bLimitBwd <-> Channel 8/Rotation Bwd Limit In
//     PlcTask Inputs/GVL.astAxes[5].stInputs.bLimitFwd <-> Channel 7/Rotation Fwd Limit In
//     PlcTask Inputs/GVL.astAxes[6].stInputs.bLimitBwd <-> Channel 2/Horizontal Bwd Limit In
//     PlcTask Inputs/GVL.astAxes[6].stInputs.bLimitFwd <-> Channel 1/Horizontal Fwd Limit In
//     PlcTask Inputs/GVL.astAxes[7].stInputs.bLimitBwd <-> Channel 4/Vertical Z1 Bwd Limit In
//     PlcTask Inputs/GVL.astAxes[8].stInputs.bLimitBwd <-> Channel 6/Vertical Z2 Bwd Limit In
//     PlcTask Inputs/GVL.astAxes[7].stInputs.bLimitFwd <-> Channel 3/Vertical Z1 Fwd Limit In
//     PlcTask Inputs/GVL.astAxes[8].stInputs.bLimitFwd <-> Channel 5/Vertical Z2 Fwd Limit In
//   tc_project_app Instance <-> Device 1 (EtherCAT)/Term 27 (EK1100)/EL6910-(04)
//     PlcTask Inputs/GVL_Safety.LocalMode <-> StandardInputs/Standard Out Var 26
//     PlcTask Inputs/GVL_Safety.ResetPossibleAndPressed <-> StandardInputs/Standard Out Var 25
//     PlcTask Inputs/GVL_Safety.UnoccupiedMode <-> StandardInputs/Standard Out Var 27
//     PlcTask Inputs/GVL_Safety.stSafetyData.SafetyGroups[1].Diag <-> TwinSAFE Group Info Data/Alias_Decouple Info Data/Diag
//     PlcTask Inputs/GVL_Safety.stSafetyData.SafetyGroups[1].Status <-> TwinSAFE Group Info Data/Alias_Decouple Info Data/State
//     PlcTask Inputs/GVL_Safety.stSafetyData.aSafetyFBS[10].Diag <-> Function Block Info Data/Main_Prog.ESTOPS.FBMon_StateValid Info Data/Diag
//     PlcTask Inputs/GVL_Safety.stSafetyData.aSafetyFBS[10].State <-> Function Block Info Data/Main_Prog.ESTOPS.FBMon_StateValid Info Data/State
//     PlcTask Inputs/GVL_Safety.stSafetyData.aSafetyFBS[11].State <-> Function Block Info Data/Main_Prog.ESTOPS.FBRs_ResetToAxDrives Info Data/State
//     PlcTask Inputs/GVL_Safety.stSafetyData.aSafetyFBS[1].Diag <-> Function Block Info Data/OpMode.DeviceMonitoring.FBMon_LightCurtain Info Data/Diag
//     PlcTask Inputs/GVL_Safety.stSafetyData.aSafetyFBS[1].State <-> Function Block Info Data/OpMode.DeviceMonitoring.FBMon_LightCurtain Info Data/State
//     PlcTask Inputs/GVL_Safety.stSafetyData.aSafetyFBS[2].Diag <-> Function Block Info Data/OpMode.DeviceMonitoring.FBMon_Searched Info Data/Diag
//     PlcTask Inputs/GVL_Safety.stSafetyData.aSafetyFBS[2].State <-> Function Block Info Data/OpMode.DeviceMonitoring.FBMon_Searched Info Data/State
//     PlcTask Inputs/GVL_Safety.stSafetyData.aSafetyFBS[3].Diag <-> Function Block Info Data/OpMode.DeviceMonitoring.FBMon_LocalMode_Disable Info Data/Diag
//     PlcTask Inputs/GVL_Safety.stSafetyData.aSafetyFBS[3].State <-> Function Block Info Data/OpMode.DeviceMonitoring.FBMon_LocalMode_Disable Info Data/State
//     PlcTask Inputs/GVL_Safety.stSafetyData.aSafetyFBS[4].Diag <-> Function Block Info Data/OpMode.OperationModes.OpMode Info Data/Diag
//     PlcTask Inputs/GVL_Safety.stSafetyData.aSafetyFBS[4].State <-> Function Block Info Data/OpMode.OperationModes.OpMode Info Data/State
//     PlcTask Inputs/GVL_Safety.stSafetyData.aSafetyFBS[5].Diag <-> Function Block Info Data/Main_Prog.DeviceMonitoring.FBMon_EStopsCloche Info Data/Diag
//     PlcTask Inputs/GVL_Safety.stSafetyData.aSafetyFBS[5].State <-> Function Block Info Data/Main_Prog.DeviceMonitoring.FBMon_EStopsCloche Info Data/State
//     PlcTask Inputs/GVL_Safety.stSafetyData.aSafetyFBS[6].Diag <-> Function Block Info Data/Main_Prog.DeviceMonitoring.FBMon_EStopsSample Info Data/Diag
//     PlcTask Inputs/GVL_Safety.stSafetyData.aSafetyFBS[6].State <-> Function Block Info Data/Main_Prog.DeviceMonitoring.FBMon_EStopsSample Info Data/State
//     PlcTask Inputs/GVL_Safety.stSafetyData.aSafetyFBS[7].Diag <-> Function Block Info Data/Main_Prog.DeviceMonitoring.FBMon_EStopsRear Info Data/Diag
//     PlcTask Inputs/GVL_Safety.stSafetyData.aSafetyFBS[7].State <-> Function Block Info Data/Main_Prog.DeviceMonitoring.FBMon_EStopsRear Info Data/State
//     PlcTask Inputs/GVL_Safety.stSafetyData.aSafetyFBS[8].Diag <-> Function Block Info Data/Main_Prog.DeviceMonitoring.FBMon_EStopPanel Info Data/Diag
//     PlcTask Inputs/GVL_Safety.stSafetyData.aSafetyFBS[8].State <-> Function Block Info Data/Main_Prog.DeviceMonitoring.FBMon_EStopPanel Info Data/State
//     PlcTask Inputs/GVL_Safety.stSafetyData.aSafetyFBS[9].Diag <-> Function Block Info Data/Main_Prog.ESTOPS.FBMon_EStopsCombined Info Data/Diag
//     PlcTask Inputs/GVL_Safety.stSafetyData.aSafetyFBS[9].State <-> Function Block Info Data/Main_Prog.ESTOPS.FBMon_EStopsCombined Info Data/State
//     PlcTask Inputs/GVL_Safety.stSafetyData.bStopAllMotion <-> StandardInputs/Standard Out Var 29
//     PlcTask Inputs/PLC_SAFETY_LOGIC.EStop1_ChA <-> Connection Info Data/Message_10 Info Data/Input Safe Data EStop1_ChA
//     PlcTask Inputs/PLC_SAFETY_LOGIC.EStop2_ChA <-> Connection Info Data/Message_10 Info Data/Input Safe Data EStop2_ChA
//     PlcTask Inputs/PLC_SAFETY_LOGIC.EStop3_ChA <-> Connection Info Data/Message_11 Info Data/Input Safe Data EStop3_ChA
//     PlcTask Inputs/PLC_SAFETY_LOGIC.EStop4_ChA <-> Connection Info Data/Message_12 Info Data/Input Safe Data EStop4_ChA
//     PlcTask Inputs/PLC_SAFETY_LOGIC.EStop5_ChA <-> Connection Info Data/Message_12 Info Data/Input Safe Data EStop5_ChA
//     PlcTask Inputs/PLC_SAFETY_LOGIC.EStop6_ChA <-> Connection Info Data/Message_13 Info Data/Input Safe Data EStop6_ChA
//     PlcTask Inputs/PLC_SAFETY_LOGIC.EStop7_ChA <-> Connection Info Data/Message_7 Info Data/Input Safe Data EStop7_ChA
//     PlcTask Inputs/PLC_SAFETY_LOGIC.EStop1_ChB <-> Connection Info Data/Message_10 Info Data/Input Safe Data EStop1_ChB
//     PlcTask Inputs/PLC_SAFETY_LOGIC.EStop2_ChB <-> Connection Info Data/Message_10 Info Data/Input Safe Data EStop2_ChB
//     PlcTask Inputs/PLC_SAFETY_LOGIC.EStop3_ChB <-> Connection Info Data/Message_11 Info Data/Input Safe Data EStop3_ChB
//     PlcTask Inputs/PLC_SAFETY_LOGIC.EStop4_ChB <-> Connection Info Data/Message_12 Info Data/Input Safe Data EStop4_ChB
//     PlcTask Inputs/PLC_SAFETY_LOGIC.EStop5_ChB <-> Connection Info Data/Message_12 Info Data/Input Safe Data EStop5_ChB
//     PlcTask Inputs/PLC_SAFETY_LOGIC.EStop6_ChB <-> Connection Info Data/Message_13 Info Data/Input Safe Data EStop6_ChB
//     PlcTask Inputs/PLC_SAFETY_LOGIC.EStop7_ChB <-> Connection Info Data/Message_7 Info Data/Input Safe Data EStop7_ChB
//     PlcTask Inputs/PLC_SAFETY_LOGIC.LightCurtain_ChA <-> Connection Info Data/Message_17 Info Data/Input Safe Data LightCurtain_ChA
//     PlcTask Inputs/PLC_SAFETY_LOGIC.LightCurtain_ChB <-> Connection Info Data/Message_17 Info Data/Input Safe Data LightCurtain_ChB
//     PlcTask Inputs/PLC_SAFETY_LOGIC.localModeButton_Pressed <-> Connection Info Data/Message_14 Info Data/Input Safe Data LocalMode_Enable
//     PlcTask Inputs/Rotation.BC1_Error <-> Connection Info Data/Message_17 Info Data/Input Safe Data BrakeChecker1_Error
//     PlcTask Inputs/Rotation.BC2_Error <-> Connection Info Data/Message_17 Info Data/Input Safe Data BrakeChecker2_Error
//     PlcTask Inputs/Rotation.Brake1State <-> StandardInputs/Standard Out Var 34
//     PlcTask Inputs/Rotation.Brake2State <-> StandardInputs/Standard Out Var 35
//     PlcTask Inputs/Rotation.Brake1Valid <-> StandardInputs/Standard Out Var 36
//     PlcTask Inputs/Rotation.Brake2Valid <-> StandardInputs/Standard Out Var 37
//     PlcTask Inputs/Rotation.RotationSTOState <-> StandardInputs/Standard Out Var 41
//     PlcTask Inputs/Rotation.SBC_FailsafeFault <-> Connection Info Data/Message_18 Info Data/Input Safe Data FailSafeOutput
//     PlcTask Inputs/Rotation.bInBrakeTestMode <-> StandardInputs/Standard Out Var 28
//     PlcTask Outputs/GVL_Safety.stSafetyData.SafetyGroups[1].AckGroup <-> StandardOutputs/Standard In Var 20
//     PlcTask Outputs/GVL_Safety.stSafetyData.SafetyGroups[1].RunGroup <-> StandardOutputs/Standard In Var 21
//     PlcTask Outputs/Rotation.BrakeReset <-> StandardOutputs/Standard In Var 24
//     PlcTask Outputs/Rotation.FinishBrakeTesting <-> StandardOutputs/Standard In Var 42
//     PlcTask Outputs/Rotation.ManualReleaseBrake1 <-> StandardOutputs/Standard In Var 38
//     PlcTask Outputs/Rotation.ManualReleaseBrake2 <-> StandardOutputs/Standard In Var 40
//     PlcTask Outputs/Rotation.RunBrake1Test <-> StandardOutputs/Standard In Var 32
//     PlcTask Outputs/Rotation.RunBrake2Test <-> StandardOutputs/Standard In Var 33
//   tc_project_app Instance <-> Device 1 (EtherCAT)/Term 70 (AX8640-0000-0103)/Drive 71 (AX8206-0210-0104)
//     PlcTask Inputs/GVL_Safety.stSafetyData.SafetyGroups[2].Diag <-> Device (Safety)/Group Info Data/ChA_ChB_Connection_Input Info Data/Diag
//     PlcTask Inputs/GVL_Safety.stSafetyData.SafetyGroups[2].Status <-> Device (Safety)/Group Info Data/ChA_ChB_Connection_Input Info Data/State
//     PlcTask Inputs/Rotation.Brake1TimeRemaining_RAW <-> Device (Safety)/Standard Inputdata/Standard Out Var 19
//     PlcTask Inputs/Rotation.Brake2TimeRemaining_RAW <-> Device (Safety)/Standard Inputdata/Standard Out Var 20
//     PlcTask Inputs/Rotation.iQ_Current <-> Ch A/Ch A TorqueControl Inputs/Iq actual
//     PlcTask Outputs/GVL_Safety.stSafetyData.SafetyGroups[2].AckGroup <-> Device (Safety)/Standard Outputdata/Standard In Var 3
//     PlcTask Outputs/GVL_Safety.stSafetyData.SafetyGroups[2].RunGroup <-> Device (Safety)/Standard Outputdata/Standard In Var 2
//   tc_project_app Instance <-> Device 1 (EtherCAT)/Term 70 (AX8640-0000-0103)/Drive 74 (AX8206-0210-0104)
//     PlcTask Inputs/GVL_Safety.stSafetyData.SafetyGroups[3].Diag <-> Device (Safety)/Group Info Data/ChA_ChB_Connection_Input Info Data/Diag
//     PlcTask Inputs/GVL_Safety.stSafetyData.SafetyGroups[3].Status <-> Device (Safety)/Group Info Data/ChA_ChB_Connection_Input Info Data/State
//     PlcTask Outputs/GVL_Safety.stSafetyData.SafetyGroups[3].AckGroup <-> Device (Safety)/Standard Outputdata/Standard In Var 3
//     PlcTask Outputs/GVL_Safety.stSafetyData.SafetyGroups[3].RunGroup <-> Device (Safety)/Standard Outputdata/Standard In Var 2
//   tc_project_app Instance <-> NC-Task 1 SAF/Axes/Combined Vertical
//     PlcTask Inputs/GVL.astAxes[9].Axis.NcToPlc <-> Outputs/ToPlc
//     PlcTask Outputs/GVL.astAxes[9].Axis.PlcToNc <-> Inputs/FromPlc
//   tc_project_app Instance <-> NC-Task 1 SAF/Axes/Combined Vertical Calibration
//     PlcTask Inputs/GVL.astAxes[25].Axis.NcToPlc <-> Outputs/ToPlc
//     PlcTask Outputs/GVL.astAxes[25].Axis.PlcToNc <-> Inputs/FromPlc
//   tc_project_app Instance <-> NC-Task 1 SAF/Axes/Combined Vertical Sample
//     PlcTask Inputs/GVL.astAxes[26].Axis.NcToPlc <-> Outputs/ToPlc
//     PlcTask Outputs/GVL.astAxes[26].Axis.PlcToNc <-> Inputs/FromPlc
//   tc_project_app Instance <-> NC-Task 1 SAF/Axes/Combined Vertical Virtual
//     PlcTask Inputs/GVL.astAxes[27].Axis.NcToPlc <-> Outputs/ToPlc
//     PlcTask Outputs/Combined_Vertical_Virtual.EncoderPosition <-> Enc/Inputs/In/nDataIn1
//     PlcTask Outputs/GVL.astAxes[27].Axis.PlcToNc <-> Inputs/FromPlc
//   tc_project_app Instance <-> NC-Task 1 SAF/Axes/Delta
//     PlcTask Inputs/GVL.astAxes[17].Axis.NcToPlc <-> Outputs/ToPlc
//     PlcTask Outputs/GVL.astAxes[17].Axis.PlcToNc <-> Inputs/FromPlc
//     PlcTask Outputs/Tau.EncoderPosition_delta <-> Enc/Inputs/In/nDataIn1
//   tc_project_app Instance <-> NC-Task 1 SAF/Axes/Detector Offset Angled
//     PlcTask Inputs/GVL.astAxes[12].Axis.NcToPlc <-> Outputs/ToPlc
//     PlcTask Outputs/GVL.astAxes[12].Axis.PlcToNc <-> Inputs/FromPlc
//   tc_project_app Instance <-> NC-Task 1 SAF/Axes/Detector Offset Parallel
//     PlcTask Inputs/GVL.astAxes[13].Axis.NcToPlc <-> Outputs/ToPlc
//     PlcTask Outputs/GVL.astAxes[13].Axis.PlcToNc <-> Inputs/FromPlc
//   tc_project_app Instance <-> NC-Task 1 SAF/Axes/Detector Radius
//     PlcTask Inputs/GVL.astAxes[19].Axis.NcToPlc <-> Outputs/ToPlc
//     PlcTask Outputs/Drad.EncoderPosition_DetectorArcRadius <-> Enc/Inputs/In/nDataIn1
//     PlcTask Outputs/GVL.astAxes[19].Axis.PlcToNc <-> Inputs/FromPlc
//   tc_project_app Instance <-> NC-Task 1 SAF/Axes/Detector Radius External
//     PlcTask Inputs/GVL.astAxes[10].Axis.NcToPlc <-> Outputs/ToPlc
//     PlcTask Outputs/Drad_External.EncoderPosition <-> Enc/Inputs/In/nDataIn1
//     PlcTask Outputs/GVL.astAxes[10].Axis.PlcToNc <-> Inputs/FromPlc
//   tc_project_app Instance <-> NC-Task 1 SAF/Axes/Detector Radius Internal
//     PlcTask Inputs/GVL.astAxes[11].Axis.NcToPlc <-> Outputs/ToPlc
//     PlcTask Outputs/Drad_Internal.EncoderPosition <-> Enc/Inputs/In/nDataIn1
//     PlcTask Outputs/GVL.astAxes[11].Axis.PlcToNc <-> Inputs/FromPlc
//   tc_project_app Instance <-> NC-Task 1 SAF/Axes/Detector Tank Internal Offset Angle
//     PlcTask Inputs/GVL.astAxes[14].Axis.NcToPlc <-> Outputs/ToPlc
//     PlcTask Outputs/Dtank_Internal_Offset_Angle.EncoderPosition <-> Enc/Inputs/In/nDataIn1
//     PlcTask Outputs/GVL.astAxes[14].Axis.PlcToNc <-> Inputs/FromPlc
//   tc_project_app Instance <-> NC-Task 1 SAF/Axes/Detector Tank Length
//     PlcTask Inputs/GVL.astAxes[15].Axis.NcToPlc <-> Outputs/ToPlc
//     PlcTask Outputs/GVL.astAxes[15].Axis.PlcToNc <-> Inputs/FromPlc
//   tc_project_app Instance <-> NC-Task 1 SAF/Axes/Detector Tank Pivot To Window
//     PlcTask Inputs/GVL.astAxes[16].Axis.NcToPlc <-> Outputs/ToPlc
//     PlcTask Outputs/GVL.astAxes[16].Axis.PlcToNc <-> Inputs/FromPlc
//   tc_project_app Instance <-> NC-Task 1 SAF/Axes/Horizontal Calibration
//     PlcTask Inputs/GVL.astAxes[28].Axis.NcToPlc <-> Outputs/ToPlc
//     PlcTask Outputs/GVL.astAxes[28].Axis.PlcToNc <-> Inputs/FromPlc
//   tc_project_app Instance <-> NC-Task 1 SAF/Axes/Horizontal Sample
//     PlcTask Inputs/GVL.astAxes[29].Axis.NcToPlc <-> Outputs/ToPlc
//     PlcTask Outputs/GVL.astAxes[29].Axis.PlcToNc <-> Inputs/FromPlc
//   tc_project_app Instance <-> NC-Task 1 SAF/Axes/Horizontal Virtual
//     PlcTask Inputs/GVL.astAxes[30].Axis.NcToPlc <-> Outputs/ToPlc
//     PlcTask Outputs/GVL.astAxes[30].Axis.PlcToNc <-> Inputs/FromPlc
//     PlcTask Outputs/Horizontal_Virtual.EncoderPosition <-> Enc/Inputs/In/nDataIn1
//   tc_project_app Instance <-> NC-Task 1 SAF/Axes/Horizontal Z Translation
//     PlcTask Inputs/GVL.astAxes[6].Axis.NcToPlc <-> Outputs/ToPlc
//     PlcTask Outputs/GVL.astAxes[6].Axis.PlcToNc <-> Inputs/FromPlc
//   tc_project_app Instance <-> NC-Task 1 SAF/Axes/M1 - South
//     PlcTask Inputs/GVL.astAxes[1].Axis.NcToPlc <-> Outputs/ToPlc
//     PlcTask Outputs/GVL.astAxes[1].Axis.PlcToNc <-> Inputs/FromPlc
//   tc_project_app Instance <-> NC-Task 1 SAF/Axes/M2 - North
//     PlcTask Inputs/GVL.astAxes[2].Axis.NcToPlc <-> Outputs/ToPlc
//     PlcTask Outputs/GVL.astAxes[2].Axis.PlcToNc <-> Inputs/FromPlc
//   tc_project_app Instance <-> NC-Task 1 SAF/Axes/M3 - West
//     PlcTask Inputs/GVL.astAxes[3].Axis.NcToPlc <-> Outputs/ToPlc
//     PlcTask Outputs/GVL.astAxes[3].Axis.PlcToNc <-> Inputs/FromPlc
//   tc_project_app Instance <-> NC-Task 1 SAF/Axes/M4 - East
//     PlcTask Inputs/GVL.astAxes[4].Axis.NcToPlc <-> Outputs/ToPlc
//     PlcTask Outputs/GVL.astAxes[4].Axis.PlcToNc <-> Inputs/FromPlc
//   tc_project_app Instance <-> NC-Task 1 SAF/Axes/Measurement Angle
//     PlcTask Inputs/GVL.astAxes[20].Axis.NcToPlc <-> Outputs/ToPlc
//     PlcTask Outputs/Drad.EncoderPosition_MeasurementAngle <-> Enc/Inputs/In/nDataIn1
//     PlcTask Outputs/GVL.astAxes[20].Axis.PlcToNc <-> Inputs/FromPlc
//   tc_project_app Instance <-> NC-Task 1 SAF/Axes/Measurement Angle Offset
//     PlcTask Inputs/GVL.astAxes[21].Axis.NcToPlc <-> Outputs/ToPlc
//     PlcTask Outputs/GVL.astAxes[21].Axis.PlcToNc <-> Inputs/FromPlc
//   tc_project_app Instance <-> NC-Task 1 SAF/Axes/Rotation
//     PlcTask Inputs/GVL.astAxes[5].Axis.NcToPlc <-> Outputs/ToPlc
//     PlcTask Outputs/GVL.astAxes[5].Axis.PlcToNc <-> Inputs/FromPlc
//   tc_project_app Instance <-> NC-Task 1 SAF/Axes/Rotation Calibration
//     PlcTask Inputs/GVL.astAxes[22].Axis.NcToPlc <-> Outputs/ToPlc
//     PlcTask Outputs/GVL.astAxes[22].Axis.PlcToNc <-> Inputs/FromPlc
//   tc_project_app Instance <-> NC-Task 1 SAF/Axes/Rotation Sample
//     PlcTask Inputs/GVL.astAxes[24].Axis.NcToPlc <-> Outputs/ToPlc
//     PlcTask Outputs/GVL.astAxes[24].Axis.PlcToNc <-> Inputs/FromPlc
//   tc_project_app Instance <-> NC-Task 1 SAF/Axes/Rotation Virtual
//     PlcTask Inputs/GVL.astAxes[23].Axis.NcToPlc <-> Outputs/ToPlc
//     PlcTask Outputs/GVL.astAxes[23].Axis.PlcToNc <-> Inputs/FromPlc
//     PlcTask Outputs/Rotation_Virtual.EncoderPosition <-> Enc/Inputs/In/nDataIn1
//   tc_project_app Instance <-> NC-Task 1 SAF/Axes/Tau
//     PlcTask Inputs/GVL.astAxes[18].Axis.NcToPlc <-> Outputs/ToPlc
//     PlcTask Outputs/GVL.astAxes[18].Axis.PlcToNc <-> Inputs/FromPlc
//     PlcTask Outputs/Tau.EncoderPosition_tau <-> Enc/Inputs/In/nDataIn1
//   tc_project_app Instance <-> NC-Task 1 SAF/Axes/Vertical Y1
//     PlcTask Inputs/GVL.astAxes[7].Axis.NcToPlc <-> Outputs/ToPlc
//     PlcTask Outputs/GVL.astAxes[7].Axis.PlcToNc <-> Inputs/FromPlc
//   tc_project_app Instance <-> NC-Task 1 SAF/Axes/Vertical Y2
//     PlcTask Inputs/GVL.astAxes[8].Axis.NcToPlc <-> Outputs/ToPlc
//     PlcTask Outputs/GVL.astAxes[8].Axis.PlcToNc <-> Inputs/FromPlc

CONFIGURATION tc_project_app
    RESOURCE PLC ON TwinCAT3
        TASK PlcTask(INTERVAL := T#2ms, PRIORITY := 10);
        PROGRAM MAIN WITH PlcTask : MAIN;
    END_RESOURCE
END_CONFIGURATION

// ---- DUTs/E_RotationBrakeCheckerState.TcDUT
{attribute 'qualified_only'}
{attribute 'strict'}
{attribute 'to_string'}
TYPE E_RotationBrakeCheckerState :
(
	init,
    Start_Brake_Test,
    Check_Drive_Mode,
    Check_Drive_Mode_To_Op,
    Set_Brake_Mode,
    Set_Brake_Mode_To_Op,
    Check_Brake_Mode,
    Check_Brake_Mode_To_Op,
    Reset_Axis,
    Confirm_STO_State,
    Enable_Motor,
    Wait_For_Test_Trigger,
    Brake_Disengage_Delay,
    Brake_Test_Triggered,
    Brake_Testing_Underway,
    In_Operation,
    Error,
    Finishing_Brake_Test
);
END_TYPE

// ---- DUTs/ST_AxisSpg.TcDUT
TYPE ST_AxisSpg :
STRUCT
    axisID : UINT;
    spgEnable : MC_ExtSetPointGenEnable;
    spgDisable : MC_ExtSetPointGenDisable;
    position : LREAL;
    velocity : LREAL;
    direction : DINT;
END_STRUCT
END_TYPE

// ---- DUTs/ST_DefaultVals.TcDUT
TYPE ST_DefaultVals :
STRUCT
    axisID : UINT;
    defaultPosition : LREAL;
    mcSetPosition : MC_SetPosition;
    deviation : LREAL;
END_STRUCT
END_TYPE

// ---- POUs/Application_Specific/Applications/eState_INTER.TcDUT
{attribute 'qualified_only'}
{attribute 'strict'}
{attribute 'to_string'}
TYPE eState_INTER :
(
	init :=0,
    setPositions :=1,
    checkSetPositions:=2,
    alignKinematics:=3,
    checkAlignKinematics:=4,
    enableSPG:=5,
    checkEnableSPG:=6,
    disableSPG:=7,
    checkDisableSPG:=8,
    operation:=9,
    startRecovery:=10,
    recoveryDefaultPosition:=11,
    waitForRecovery:=12,
    fixRotation:=13,
    error:=999,
    safetyError:=666,
    none:=1000,
    localModeDisabled:=14
);
END_TYPE

// ---- POUs/Application_Specific/Applications/eState_Vertical.TcDUT
{attribute 'qualified_only'}
{attribute 'strict'}
TYPE eState_Vertical :
(
	init := 0,
    checkPosition := 1,
    setPosition := 2,
    enableSpg := 3,
    confirmEnableSpg := 4,
    disableSpg := 5,
    confirmDisableSpg :=6,
    operation :=7
    
);
END_TYPE

// ---- tc_mca_std_lib/DUTs/Axis_Structures/ST_AxisDescription.TcDUT
TYPE ST_AxisDescription :
STRUCT
    sAxisName : STRING(nMAX_AXIS_NAME);
    nUnit: BYTE; //Code for the axis base unit (like m or degree)
    nPrefix: BYTE; //Exponent defining unit prefix, e.g. 3 for k(kilo)
    bIsPseudoAxis: BOOL; //Axis is a non-standard axis with application-specific handling
    eEncoderType: E_EncoderTypeClass;
    eHomeSwitchType: E_HomeSwitchTypeClass;
    eMotorType: E_MotorTypeClass;
END_STRUCT
END_TYPE

// ---- tc_mca_std_lib/DUTs/Axis_Structures/ST_AxisStatus.TcDUT
TYPE ST_AxisStatus :
STRUCT
    //Outputs & Status
    bAxisInitialized: BOOL := FALSE; //True when all parameters from actReadMcParameters are valid
    bEnabled: BOOL; //Axis drive enabled
    bCommandAborted: BOOL; //Command aborted output of the eCommand function blocks
    bBusy: BOOL; //Axis busy (eCommand function block is active)
    bDone: BOOL; //Last eCommand function block executed successfully;
    //bDone will also be set with the InGear and InVelocity outputs
    //When InVelocity is set, fbMoveVelocity is still acitve, which is reflected by the bBusy status
    bInVelocity: BOOL; //MC_MoveVelocity has reached target velocity; will stay true until the movement stops
    bHomed: BOOL; //Axis homed
    bMoving: BOOL; //Moving state from the NC
    bMovingForward: BOOL; //Moving forward indicator from NC
    bMovingBackward: BOOL; //Moving backward indicator from NC
    bInTargetPosition: BOOL; //In target position bit from AxisStatus()
    bFwEnabled: BOOL; //Positive movement of axis is enabled/disabled
    bBwEnabled: BOOL; //Negative movement of axis is enabled/disabled
    bInterlockedFwd: BOOL; //Axis interlocked in the postive direction
    bInterlockedBwd: BOOL; //Axis interlocked in the negative direction
    bGeared: BOOL; //Axis is an active slave
    bCoupledGear1: BOOL;
    bCoupledGear2: BOOL;
    bCoupledGear3: BOOL;
    bCoupledGear4: BOOL;
    fActPosition: LREAL; //Actual position value
    nEncoderRawCounter AT %I*: UDINT; //Raw encoder counter value
    nStepperDriveCounter AT %I*: UDINT; //Raw internal counter from stepper drive
    fActVelocity: LREAL; //Actual velocity
    bError: BOOL; //Motion function block has produced error (NC drive not necessarily in error state)
    nErrorID: UDINT; //Last motion function block errorID or NC errorID
END_STRUCT
END_TYPE

// ---- tc_mca_std_lib/DUTs/Axis_Structures/ST_AxisStruct.TcDUT
TYPE ST_AxisStruct :
STRUCT
    stControl: ST_AxisControl;
    stStatus: ST_AxisStatus;
    stConfig: ST_AxisConfig;
    stError: ST_AxisError;
    stInputs: ST_AxisInputs;
	stDescription: ST_AxisDescription;
	stSafety : ST_AxisSafety;
    //The NC axis link to the hardware that is controlling
    Axis: AXIS_REF;
END_STRUCT
END_TYPE

// ---- tc_mca_std_lib/DUTs/E_HomingRoutines.TcTLEO
{attribute 'qualified_only'}
{attribute 'strict'}
TYPE E_HomingRoutines :
(
    eNoHoming := 0,

    //0X: LIMIT Switch
    //Home to bBwdLimit, record position on first approach
    eHomeToLimit_Bwd := 1,
    //Home to bFwdLimit, record position on first approach
    eHomeToLimit_Fwd := 2,
    //Find bBwdLimit (using towardsCam speed), then reverse direction looking FOR falling edge (using fromCam speed)
    //eHomeToLimit_Bwd_2Speeds := 3,
    //Find bFwdLimit (using towardsCam speed), then reverse direction looking for falling edge (using fromCam speed)
    //eHomeToLimit_Fwd_2Speeds := 4,

    //1X: Home Sensor
    //Home to bHome in Bwd direction (will reverse direction if limit hit), record position on first approach
    eHomeToRef_Bwd := 11,
    //Home to bHome in Fwd direction (will reverse direction if limit hit), record position on first approach
    eHomeToRef_Fwd := 12,
    //Find bHome in Bwd direction (using towardsCam speed) then reverse direction looking for falling edge (using fromCam speed), will reverse direction if limit hit
    //eHomeToRef_Bwd_2Speeds := 13,
    //Find bHome in Fwd direction (using towardsCam speed) then reverse direction looking for falling edge (using fromCam speed), will reverse direction if limit hit
    //eHomeToRef_Fwd_2Speeds := 14,

    //2X: Enc Pulse
    //Home to EncRefPulse in Bwd direction (used for single turn rotary axis without limit switches)
    eHomeToEncPulse_Bwd := 21,
    //Home to EncRefPulse in Fwd direction (used for single turn rotary axis without limit switches)
    eHomeToEncPulse_Fwd := 22,
    //Home to EncRefPulse via bBwdLimit (using towardsCam speed), then reverse direction looking for falling edge on ref pulse (using fromCam speed)
    eHomeToEncPulse_viaBwdLimit := 23,
    //Home to EncRefPulse via bFwdLimit (using towardsCam speed), then reverse direction looking for falling edge on ref pulse (using fromCam speed)
    eHomeToEncPulse_viaFwdLimit := 24,

    //3X: Home To Mechanical Block (Lag based StepBlockDetection)
    //Home towards a mechanical block in Bwd direction
    eHomeToBlock_Bwd := 30,
    //Home towards a mechanical block in Fwd direction
    eHomeToBlock_Fwd := 31,

    //9X: Software
    eHomeDirect := 90 //Set position directly to fHomePosition
) := eNoHoming;
END_TYPE

// ---- tc_mca_std_lib/DUTs/E_MotorTypeClass.TcDUT
TYPE E_MotorTypeClass :
(
    eVirtualMotor := 0, //Axis is Virtual
    eStepperMotor := 1, //Axis based on a stepper motor
    eDcMotor := 2, //Axis based on a brushed DC motor
    eBldcMotor := 3, //Axis based on a BLDC motor
    eAsyncMotor := 4, //Axis based on a three phase asynchronous motor
    eSyncMotor := 5 //Axis based on a three phase synchronous motor
) := eVirtualMotor;
END_TYPE

// ---- tc_mca_std_lib/DUTs/E_EncoderTypeClass.TcDUT
TYPE E_EncoderTypeClass :
(
    eNoEncoder := 0,
    eIncrementalEncoder := 1,
    eAbsoluteEncoder := 2
) := eNoEncoder;
END_TYPE

// ---- tc_mca_std_lib/DUTs/E_HomeSwitchTypeClass.TcDUT
TYPE E_HomeSwitchTypeClass:
(
    eNoSwitch := 0, //no physical switch for homing present
    eHomeSwitchPresent := 1, //dedicated homing switch present
    eUseBwdLimit := 2, //Bwd limit switch is used as a homing switch
    eUseFwdLimit := 3 //Fwd limit switch is used as a homing switch
) := eNoSwitch;
END_TYPE

// ---- tc_mca_std_lib/DUTs/Safety Status/E_SafetyFbState.TcDUT
TYPE E_SafetyFbState :
(
	RUN := 1,
    STOP :=2,
    SAFE :=3,
    ERROR := 4,
    RESET := 5,
    START := 6,
    ERRORDELAY := 7,
    DELAYOUT := 8,
    FUNCTEST := 9
);
END_TYPE

// ---- tc_mca_std_lib/DUTs/Safety Status/E_SafetyFbType.TcDUT
{attribute 'qualified_only'}
{attribute 'strict'}
TYPE E_SafetyFbType :
(
	Unassigned := 0,
    FB_Mon := 1,
    FB_OpMode := 2,
    FB_RS :=3,
    FB_SR :=4,
    FB_EDM :=5
);
END_TYPE

// ---- tc_mca_std_lib/DUTs/Safety Status/E_SafetyGroupState.TcDUT
TYPE E_SafetyGroupState :
(
	RUN := 1,
    STOP := 2,
    ERROR := 4,
    RESET := 5,
    START := 6,
    STOPERROR := 7,
    DEACTIVE := 16,
    WAITCOMERROR := 17
);
END_TYPE

// ---- tc_mca_std_lib/DUTs/Safety Status/ST_SafetyAliasInput.TcDUT
TYPE ST_SafetyAliasInput :
STRUCT
	sName : STRING; //Name descriptor for the safety output
    bState : BOOL;
END_STRUCT
END_TYPE

// ---- tc_mca_std_lib/DUTs/Safety Status/ST_SafetyData.TcDUT
TYPE ST_SafetyData :
STRUCT
	bSafetyAckReq : BOOL;   //SafetyProgram requires acknowledge

    bResetPressed : BOOL; //Read only implementation
	sBannerMessage : STRING(255); // Max string length
	bStopAllMotion AT %I* : BOOL; //Command bool to IBEX to initiate a non-ss1 stop on galil axes
	
	bSearchedAndLocked AT %I* : BOOL;
	
	aSafetyAliasOuputs : ARRAY[1..GVL_Safety.nSAFETY_OUTPUTS] OF ST_SafetyAliasOutput;
	aSafetyAliasInputs : ARRAY[1..GVL_Safety.nSAFETY_INPUTS] OF ST_SafetyAliasInput;
	aSafetyDevices : ARRAY[1..GVL_Safety.nSAFETY_DEVICES] OF ST_SafetyDevice;
    aSafetyFBS : ARRAY[1..GVL_Safety.nSAFETY_FBS] OF ST_SafetyFB;

    SafetyGroups : ARRAY[1..GVL_Safety.nSAFETY_GROUPS] OF ST_SafetyGroup;
    sInError : STRING;
    sInErrorDiag : STRING;
    sDiagMessageToUser : STRING;
    
END_STRUCT
END_TYPE

// ---- tc_mca_std_lib/DUTs/Safety Status/ST_SafetyFB.TcDUT
TYPE ST_SafetyFB :
STRUCT
    sName : STRING;
    Diag AT %I* : UINT;
    State AT %I* : USINT;
    eFbType : E_SafetyFbType;
    fbState : E_SafetyFbState;
    DiagString : STRING;
END_STRUCT
END_TYPE

// ---- tc_mca_std_lib/DUTs/Safety Status/ST_SafetyGroup.TcDUT
TYPE ST_SafetyGroup :
STRUCT
    Name : STRING;
    RunGroup AT %Q* : BOOL := TRUE; //Auto default to run state
    AckGroup AT %Q* : BOOL;
    
    Diag AT %I* : BYTE;
    Status AT %I* : BYTE;
    groupState : E_SafetyGroupState;
END_STRUCT
END_TYPE

// ---- tc_mca_std_lib/DUTs/Safety Status/ST_SafetyAliasOutput.TcDUT
TYPE ST_SafetyAliasOutput :
STRUCT
	sName : STRING; //Name descriptor for the safety output
    bState : BOOL;
END_STRUCT
END_TYPE

// ---- tc_mca_std_lib/DUTs/Safety Status/ST_SafetyProject.TcDUT
TYPE ST_SafetyProject :
STRUCT
	inRun AT %I* : BOOL;
	inError AT %I* : BOOL;
	inResetRequired AT %I* : BOOL;
	
	outAcknowledgeError AT %Q* : BOOL;
	outRunProject AT %Q* : BOOL;
	
	//ANY OTHERS?
	
END_STRUCT
END_TYPE

// ---- GVLs/GVL_APP.TcGVL
{attribute 'qualified_only'}
VAR_GLOBAL
END_VAR

VAR_GLOBAL CONSTANT
    nAXIS_NUM: UINT := 30;
    nPNEUMATIC_AXIS_NUM: UINT := 0;
END_VAR

// ---- GVLs/GVL_INTER.TcGVL
{attribute 'qualified_only'}
VAR_GLOBAL
    RUN_KINEMATICS : BOOL := FALSE;
    RUN_COUPLED_VERTICAL : BOOL := TRUE;    //DEFAULT ALWAYS ON, JUST STARTS LOGIC
    DECOUPLE_VERTICAL_AXES : BOOL;
    DISABLE_ALL_AXES : BOOL;
    ENABLE_ALL_AXES : BOOL;
    RESET_ALL : BOOL;
    ACKNOWLEDGE_LOGIC_ERROR : BOOL;
    REMOTE_RESET : BOOL;
    
    
    REINITIALISE : BOOL;
    FINISH_REINITIALISE : BOOL;
    
    START_RECOVERY : BOOL;
    
    UPDATE_DEFAULTS : BOOL;
    CLEAR_ALL_DEFAULTS : BOOL;
    
    
    //STATUSES
    LIMIT_HIT : BOOL;
    OPERATIONAL : BOOL;
    NC_AXIS_ERROR : BOOL;
    REINITIALISE_IN_PROGRESS : BOOL;
    RECOVERY_IN_PROGRESS : BOOL;
    REAL_AXES_NOT_MOVING : BOOL;
    VIRTUAL_AXES_NOT_MOVING : BOOL;
    KINEMATIC_SPG_ALL_ENABLED : BOOL;
    KINEMATIC_SPG_ALL_DISABLED : BOOL;
    LOGIC_ERROR : BOOL;
    LOGIC_STATE : eState_INTER;
    LOGIC_STATE_ERROR : eState_INTER := eState_INTER.none;
	LOGIC_STATE_STR: STRING;
	LOGIC_STATE_ERROR_STR: STRING;
    SAFETY_ACK_REQUESTED : BOOL;
    RESET_REQUESTED : BOOL;
    SPEED_LIMITING : BOOL;
    //POSITIONS
    SETPOS_HORIZONTAL : LREAL;
    SETPOS_COMBINED_VERTICAL : LREAL;
    SETPOS_ROTATION : LREAL;
    SETVELO_HORIZONTAL : LREAL;
    SETVELO_COMBINED_VERTICAL : LREAL;
    SETVELO_ROTATION : LREAL;
    SETDIR_HORIZONTAL : DINT;
    SETDIR_COMBINED_VERTICAL : DINT;
    SETDIR_ROTATION : DINT;
    BRAKE_TEST_PASSED : BOOL;
    
    
    
    TARGET_MEASUREMENT_ANGLE : LREAL;
    
    INCLINOMETER_ANGLE : LREAL;
    
END_VAR

// ---- GVLs/GVL_Safety.TcGVL
{attribute 'qualified_only'}
VAR_GLOBAL
    stSafetyData : ST_SafetyData;   //Main safety data structure for project
    
    //Run_MotionSafety AT %Q* : BOOL := TRUE;
    //Run_MotionSafety_XRotAndZHor AT %Q* : BOOL:= TRUE;
    //Run_MotionSafety_Y1AndY2 AT %Q* : BOOL:= TRUE;
    //    
    //ErrorAck_MotionSafety AT %Q* : BOOL;   
    //ErrorAck_MotionSafety_XRotAndZHor AT %Q* : BOOL;    
    //ErrorAck_MotionSafety_Y1AndY2 AT %Q* : BOOL;
    
    
    
    ResetPossibleAndPressed AT %I* : BOOL;
    
    SAFETY_ACK : BOOL; //Combined safety acknowledge var
    
    LocalMode AT %I* : BOOL;
    UnoccupiedMode AT %I* : BOOL;
    LocalMode_Disabled : BOOL;
    
    fbMon_StateValid_Status AT %I* : BYTE;



    
    
   
END_VAR
VAR_GLOBAL CONSTANT
    nSAFETY_OUTPUTS: UINT := 3; //do these break with a 0 value?
    nSAFETY_INPUTS: UINT := 1; //do these break with a 0 value?
	nSAFETY_DEVICES: UINT := 1;
    nSAFETY_FBS: UINT := 15;
    nSAFETY_GROUPS: UINT := 3;
END_VAR

// ---- POUs/Application_Specific/Axes/AXIS_NAMES.TcGVL
VAR_GLOBAL CONSTANT
    
    //RAW AXES
    AXIS_SLIT_NORTH : UINT :=1;
    AXIS_SLIT_SOUTH : UINT :=2;
    AXIS_SLIT_EAST : UINT :=3;
    AXIS_SLIT_WEST : UINT :=4;
    AXIS_ROTATION : UINT:= 5; //rotation about X axis
    AXIS_HORIZONTAL_TRANSLATION : UINT :=6; //Z translation along beam
    AXIS_VERTICAL_TRANSLATION_Y1 : UINT :=7;
    AXIS_VERTICAL_TRANSLATION_Y2 : UINT :=8;
    
    //COMBINED MOTION AXES
    AXIS_COMBINED_VERTICAL : UINT :=9;
    
    
    
    //DRAD = DETECTOR RADIUS
    //DOFF = DETECTOR OFFSET
    //DTANK = DETECTOR TANK
    
    
    //UNIMPLEMENTED LIST TO WORK THROUGH
    AXIS_DRAD_EXTERNAL : UINT :=10;
    AXIS_DRAD_INTERNAL : UINT :=11;
    
    AXIS_DOFF_ANGLED : UINT :=12;
    AXIS_DOFF_PARALLEL : UINT :=13;
    
    AXIS_DTANK_INTERNAL_OFFSET_ANGLE : UINT :=14;
    
    AXIS_DTANK_LENGTH : UINT :=15;
    AXIS_DTANK_PIVOT_TO_WINDOW : UINT :=16;
    
    AXIS_DELTA : UINT :=17;
    AXIS_TAU : UINT :=18;
    
    AXIS_DRAD : UINT :=19;
    AXIS_MEASUREMENT_ANGLE : UINT :=20;
    
    AXIS_MEASUREMENT_ANGLE_OFFSET : UINT :=21;
    
    AXIS_ROTATION_CALIBRATION : UINT :=22;
    AXIS_ROTATION_VIRTUAL : UINT :=23;
    AXIS_ROTATION_SAMPLE : UINT :=24;
    
